ACTION ModeENLimk:
//屏蔽链接
Mach_Control.DT_b.FirstEmpFold:=par.iModeEN.FirstEmpFoldEN;				//首层空叠隔膜屏蔽
Mach_Control.DT_b.DP_Mode:=NOT par.iModeEN.DP_ModeEN;				//尾层空叠隔膜屏蔽
Mach_Control.DT_b.RectifydevModel:=par.iModeEN.RectifydevModelEN;			//隔膜纠偏屏蔽
Mach_Control.U.EmptyRunMode:=par.iModeEN.EmptyRunModeEN;				//空叠隔膜屏蔽
Mach_Control.U.CCD_ChosesHMI:=par.iModeEN.CCD_ChosesHMIEN;			//CCD屏蔽
Mach_Control.DT_b.DT_CCD_TwoModel:=NOT par.iModeEN.DT_CCD_TwoModelEN;		//CCD复检屏蔽
Mach_Control.DT_b.DT_Overhang:=par.iModeEN.DT_OverhangEN;				//对齐度屏蔽
Mach_Control.DT_b.DT_CellNG_TF:=NOT par.iModeEN.DT_CellNG_TFEN;				//对齐度踢废屏蔽 
Mach_Control.DT_b.DT_OHclosure:= par.iModeEN.DT_OHclosureEN;				//对齐度闭环屏蔽		ON是屏蔽
Mach_Control.DT_b.GMAngleALMsel:= par.iModeEN.GMAngleALMsel; //隔膜卷径报警屏蔽		ON是屏蔽
END_ACTION

ACTION MotionCoe_Write:

//nSlaveAddr :ARRAY[1..6] OF INT :=[1003,1008,1018,1019,1020,1021] ;     //EtherCAT支路驱动器ID

//'192.168.10.10.4.1'	EtherCat支路ID
(*
//隔膜平移地址
P2M1_Par.stDT_date.EtherCatAddr[1]:=1172;
P2M2_Par.stDT_date.EtherCatAddr[1]:=1123;
P2M3_Par.stDT_date.EtherCatAddr[1]:=1077;

//隔膜缓存地址
P2M1_Par.stDT_date.EtherCatAddr[2]:=1173;
P2M2_Par.stDT_date.EtherCatAddr[2]:=1124;
P2M3_Par.stDT_date.EtherCatAddr[2]:=1078;

//正极送片搬运平移地址
P2M1_Par.stDT_date.EtherCatAddr[3]:=1170;
P2M2_Par.stDT_date.EtherCatAddr[3]:=1121;
P2M3_Par.stDT_date.EtherCatAddr[3]:=1075;

//正极叠片搬运平移地址
P2M1_Par.stDT_date.EtherCatAddr[4]:=1171;
P2M2_Par.stDT_date.EtherCatAddr[4]:=1122;
P2M3_Par.stDT_date.EtherCatAddr[4]:=1076;

//负极送片搬运平移地址
P2M1_Par.stDT_date.EtherCatAddr[5]:=1188;
P2M2_Par.stDT_date.EtherCatAddr[5]:=1139;
P2M3_Par.stDT_date.EtherCatAddr[5]:=1093;

//负极叠片搬运平移地址
P2M1_Par.stDT_date.EtherCatAddr[6]:=1172;
P2M2_Par.stDT_date.EtherCatAddr[6]:=1140;
P2M3_Par.stDT_date.EtherCatAddr[6]:=1094;

//////////////////////////////////////////////////////////////////////一号叠台隔膜平移
FB_EcCoESdoWrite_SEPTATLine[1](
	sNetId:= '192.168.10.10.4.1', 
	nSlaveAddr:=Par.stDT_date.EtherCatAddr[1] ,   //隔膜平移
	nSubIndex:=0 , 
	nIndex:=16#2108 ,   //  平滑时间
	pSrcBuf:=ADR(Par.stDT_date.SEPTATLine_fSmoothValue[1]),       //写入参数值 
	cbBufLen:=SIZEOF(Par.stDT_date.SEPTATLine_fSmoothValue[1]),    
	bExecute:= Par.stDT_date.SEPTATLine_bWriteCoeValue[1],    
	tTimeout:= T#3S, 
	bBusy=> , 
	bError=> , 
	nErrId=> );
	
FB_EcCoESdoWrite_SEPTATLine[2](
	sNetId:='192.168.10.10.4.1', 
	nSlaveAddr:=Par.stDT_date.EtherCatAddr[1] ,   //隔膜平移
	nSubIndex:=0 , 
	nIndex:=16#2109 ,   // 平滑方式
	pSrcBuf:=ADR(Par.stDT_date.SEPTATLine_fSmoothValue[2]),       //写入参数值 
	cbBufLen:=SIZEOF(Par.stDT_date.SEPTATLine_fSmoothValue[2]),    
	bExecute:= Par.stDT_date.SEPTATLine_bWriteCoeValue[2],    
	tTimeout:= T#3S, 
	bBusy=> , 
	bError=> , 
	nErrId=> );

//平滑时间参数保存	
FB_EcCoESdoWrite_SEPTATLine[3](
	sNetId:= '192.168.10.10.4.1', 
	nSlaveAddr:=Par.stDT_date.EtherCatAddr[1] ,   //隔膜平移
	nSubIndex:=0 , 
	nIndex:=16#2108 ,   // 平滑时间
	pSrcBuf:=ADR(Par.stDT_date.wSaveCoeCode),      
	cbBufLen:=SIZEOF(Par.stDT_date.wSaveCoeCode),    
	bExecute:= Par.stDT_date.SEPTATLine_SavePara[1],    
	tTimeout:= T#3S, 
	bBusy=> , 
	bError=> , 
	nErrId=> );	
	
//平滑方式参数保存	
FB_EcCoESdoWrite_SEPTATLine[4](
	sNetId:= '192.168.10.10.4.1', 
	nSlaveAddr:=Par.stDT_date.EtherCatAddr[1] ,   //隔膜平移
	nSubIndex:=0 , 
	nIndex:=16#2109 ,   // 平滑方式
	pSrcBuf:=ADR(Par.stDT_date.wSaveCoeCode),      
	cbBufLen:=SIZEOF(Par.stDT_date.wSaveCoeCode),    
	bExecute:= Par.stDT_date.SEPTATLine_SavePara[2],    
	tTimeout:= T#3S, 
	bBusy=> , 
	bError=> , 
	nErrId=> );	

	
//////////////////////////////////////////////////////////////////////一号叠台隔膜缓存
FB_EcCoESdoWrite_SEPTATCache[1](
	sNetId:='192.168.10.10.4.1', 
	nSlaveAddr:=Par.stDT_date.EtherCatAddr[2] ,   //隔膜缓存
	nSubIndex:=0 , 
	nIndex:=16#2108 ,   //  平滑时间
	pSrcBuf:=ADR(Par.stDT_date.SEPTATCache_fSmoothValue[1]),       //写入参数值 
	cbBufLen:=SIZEOF(Par.stDT_date.SEPTATCache_fSmoothValue[1]),    
	bExecute:= Par.stDT_date.SEPTATCache_bWriteCoeValue[1],    
	tTimeout:= T#3S, 
	bBusy=> , 
	bError=> , 
	nErrId=> );
	
FB_EcCoESdoWrite_SEPTATCache[2](
	sNetId:='192.168.10.10.4.1', 
	nSlaveAddr:=Par.stDT_date.EtherCatAddr[2] ,   //隔膜缓存
	nSubIndex:=0 , 
	nIndex:=16#2109 ,   // 平滑方式
	pSrcBuf:=ADR(Par.stDT_date.SEPTATCache_fSmoothValue[2]),       //写入参数值 
	cbBufLen:=SIZEOF(Par.stDT_date.SEPTATCache_fSmoothValue[2]),    
	bExecute:= Par.stDT_date.SEPTATCache_bWriteCoeValue[2],    
	tTimeout:= T#3S, 
	bBusy=> , 
	bError=> , 
	nErrId=> );

//平滑时间参数保存	
FB_EcCoESdoWrite_SEPTATCache[3](
	sNetId:= '192.168.10.10.4.1', 
	nSlaveAddr:=Par.stDT_date.EtherCatAddr[2] ,   //隔膜缓存
	nSubIndex:=0 , 
	nIndex:=16#2108 ,   // 平滑时间
	pSrcBuf:=ADR(Par.stDT_date.wSaveCoeCode),      
	cbBufLen:=SIZEOF(Par.stDT_date.wSaveCoeCode),    
	bExecute:= Par.stDT_date.SEPTATCache_SavePara[1],    
	tTimeout:= T#3S, 
	bBusy=> , 
	bError=> , 
	nErrId=> );	
	
//平滑方式参数保存	
FB_EcCoESdoWrite_SEPTATCache[4](
	sNetId:= '192.168.10.10.4.1', 
	nSlaveAddr:=Par.stDT_date.EtherCatAddr[2] ,   //隔膜缓存
	nSubIndex:=0 , 
	nIndex:=16#2109 ,   // 平滑方式
	pSrcBuf:=ADR(Par.stDT_date.wSaveCoeCode),      
	cbBufLen:=SIZEOF(Par.stDT_date.wSaveCoeCode),    
	bExecute:= Par.stDT_date.SEPTATCache_SavePara[2],    
	tTimeout:= T#3S, 
	bBusy=> , 
	bError=> , 
	nErrId=> );	
	
	
//////////////////////////////////////////////////////////////////////正极送片搬运平移
FB_EcCoESdoWrite_AnCarryingLine[1](
	sNetId:= '192.168.10.10.4.1', 
	nSlaveAddr:=Par.stDT_date.EtherCatAddr[3] ,   //正极送片搬运平移
	nSubIndex:=0 , 
	nIndex:=16#2108 ,   //  平滑时间
	pSrcBuf:=ADR(Par.stDT_date.AnCarryingLine_fSmoothValue[1]),       //写入参数值 
	cbBufLen:=SIZEOF(Par.stDT_date.AnCarryingLine_fSmoothValue[1]),    
	bExecute:= Par.stDT_date.AnCarryingLine_bWriteCoeValue[1],    
	tTimeout:= T#3S, 
	bBusy=> , 
	bError=> , 
	nErrId=> );
	
FB_EcCoESdoWrite_AnCarryingLine[2](
	sNetId:= '192.168.10.10.4.1', 
	nSlaveAddr:=Par.stDT_date.EtherCatAddr[3]  ,   //正极送片搬运平移
	nSubIndex:=0 , 
	nIndex:=16#2109 ,   // 平滑方式
	pSrcBuf:=ADR(Par.stDT_date.AnCarryingLine_fSmoothValue[2]),       //写入参数值 
	cbBufLen:=SIZEOF(Par.stDT_date.AnCarryingLine_fSmoothValue[2]),    
	bExecute:= Par.stDT_date.AnCarryingLine_bWriteCoeValue[2],    
	tTimeout:= T#3S, 
	bBusy=> , 
	bError=> , 
	nErrId=> );

//平滑时间参数保存	
FB_EcCoESdoWrite_AnCarryingLine[3](
	sNetId:= '192.168.10.10.4.1', 
	nSlaveAddr:=Par.stDT_date.EtherCatAddr[3]  ,   //正极送片搬运平移
	nSubIndex:=0 , 
	nIndex:=16#2108 ,   // 平滑时间
	pSrcBuf:=ADR(Par.stDT_date.wSaveCoeCode),      
	cbBufLen:=SIZEOF(Par.stDT_date.wSaveCoeCode),    
	bExecute:= Par.stDT_date.AnCarryingLine_SavePara[1],    
	tTimeout:= T#3S, 
	bBusy=> , 
	bError=> , 
	nErrId=> );	
	
//平滑方式参数保存	
FB_EcCoESdoWrite_AnCarryingLine[4](
	sNetId:= '192.168.10.10.4.1', 
	nSlaveAddr:=Par.stDT_date.EtherCatAddr[3]  ,   //正极送片搬运平移
	nSubIndex:=0 , 
	nIndex:=16#2109 ,   // 平滑方式
	pSrcBuf:=ADR(Par.stDT_date.wSaveCoeCode),      
	cbBufLen:=SIZEOF(Par.stDT_date.wSaveCoeCode),    
	bExecute:= Par.stDT_date.AnCarryingLine_SavePara[2],    
	tTimeout:= T#3S, 
	bBusy=> , 
	bError=> , 
	nErrId=> );		
	
//////////////////////////////////////////////////////////////////////正极叠片搬运平移
FB_EcCoESdoWrite_AnDTCarryingLine[1](
	sNetId:='192.168.10.10.4.1', 
	nSlaveAddr:=Par.stDT_date.EtherCatAddr[4]  ,   //正极叠片搬运平移
	nSubIndex:=0 , 
	nIndex:=16#2108 ,   //  平滑时间
	pSrcBuf:=ADR(Par.stDT_date.AnDTCarryingLine_fSmoothValue[1]),       //写入参数值 
	cbBufLen:=SIZEOF(Par.stDT_date.AnDTCarryingLine_fSmoothValue[1]),    
	bExecute:= Par.stDT_date.AnDTCarryingLine_bWriteCoeValue[1],    
	tTimeout:= T#3S, 
	bBusy=> , 
	bError=> , 
	nErrId=> );
	
FB_EcCoESdoWrite_AnDTCarryingLine[2](
	sNetId:= '192.168.10.10.4.1', 
	nSlaveAddr:=Par.stDT_date.EtherCatAddr[4]  ,   //正极叠片搬运平移
	nSubIndex:=0 , 
	nIndex:=16#2109 ,   // 平滑方式
	pSrcBuf:=ADR(Par.stDT_date.AnDTCarryingLine_fSmoothValue[2]),       //写入参数值 
	cbBufLen:=SIZEOF(Par.stDT_date.AnDTCarryingLine_fSmoothValue[2]),    
	bExecute:= Par.stDT_date.AnDTCarryingLine_bWriteCoeValue[2],    
	tTimeout:= T#3S, 
	bBusy=> , 
	bError=> , 
	nErrId=> );

//平滑时间参数保存	
FB_EcCoESdoWrite_AnDTCarryingLine[3](
	sNetId:= '192.168.10.10.4.1', 
	nSlaveAddr:=Par.stDT_date.EtherCatAddr[4]  ,   //正极叠片搬运平移
	nSubIndex:=0 , 
	nIndex:=16#2108 ,   // 平滑时间
	pSrcBuf:=ADR(Par.stDT_date.wSaveCoeCode),      
	cbBufLen:=SIZEOF(Par.stDT_date.wSaveCoeCode),    
	bExecute:= Par.stDT_date.AnDTCarryingLine_SavePara[1],    
	tTimeout:= T#3S, 
	bBusy=> , 
	bError=> , 
	nErrId=> );	
	
//平滑方式参数保存	
FB_EcCoESdoWrite_AnDTCarryingLine[4](
	sNetId:= '192.168.10.10.4.1', 
	nSlaveAddr:=Par.stDT_date.EtherCatAddr[4]  ,   //正极叠片搬运平移
	nSubIndex:=0 , 
	nIndex:=16#2109 ,   // 平滑方式
	pSrcBuf:=ADR(Par.stDT_date.wSaveCoeCode),      
	cbBufLen:=SIZEOF(Par.stDT_date.wSaveCoeCode),    
	bExecute:= Par.stDT_date.AnDTCarryingLine_SavePara[2],    
	tTimeout:= T#3S, 
	bBusy=> , 
	bError=> , 
	nErrId=> );			
	
//////////////////////////////////////////////////////////////////////负极送片搬运平移
FB_EcCoESdoWrite_CaCarryingLine2[1](
	sNetId:= '192.168.10.10.4.1', 
	nSlaveAddr:=Par.stDT_date.EtherCatAddr[5]  ,   //负极送片搬运平移
	nSubIndex:=0 , 
	nIndex:=16#2108 ,   //  平滑时间
	pSrcBuf:=ADR(Par.stDT_date.CaCarryingLine2_fSmoothValue[1]),       //写入参数值 
	cbBufLen:=SIZEOF(Par.stDT_date.CaCarryingLine2_fSmoothValue[1]),    
	bExecute:= Par.stDT_date.CaCarryingLine2_bWriteCoeValue[1],    
	tTimeout:= T#3S, 
	bBusy=> , 
	bError=> , 
	nErrId=> );
	
FB_EcCoESdoWrite_CaCarryingLine2[2](
	sNetId:= '192.168.10.10.4.1', 
	nSlaveAddr:=Par.stDT_date.EtherCatAddr[5] ,   //负极送片搬运平移
	nSubIndex:=0 , 
	nIndex:=16#2109 ,   // 平滑方式
	pSrcBuf:=ADR(Par.stDT_date.CaCarryingLine2_fSmoothValue[2]),       //写入参数值 
	cbBufLen:=SIZEOF(Par.stDT_date.CaCarryingLine2_fSmoothValue[2]),    
	bExecute:= Par.stDT_date.CaCarryingLine2_bWriteCoeValue[2],    
	tTimeout:= T#3S, 
	bBusy=> , 
	bError=> , 
	nErrId=> );

//平滑时间参数保存	
FB_EcCoESdoWrite_CaCarryingLine2[3](
	sNetId:= '192.168.10.10.4.1', 
	nSlaveAddr:=Par.stDT_date.EtherCatAddr[5] ,   //负极送片搬运平移
	nSubIndex:=0 , 
	nIndex:=16#2108 ,   // 平滑时间
	pSrcBuf:=ADR(Par.stDT_date.wSaveCoeCode),      
	cbBufLen:=SIZEOF(Par.stDT_date.wSaveCoeCode),    
	bExecute:= Par.stDT_date.CaCarryingLine2_SavePara[1],    
	tTimeout:= T#3S, 
	bBusy=> , 
	bError=> , 
	nErrId=> );	
	
//平滑方式参数保存	
FB_EcCoESdoWrite_CaCarryingLine2[4](
	sNetId:='192.168.10.10.4.1', 
	nSlaveAddr:=Par.stDT_date.EtherCatAddr[5] ,   //负极送片搬运平移
	nSubIndex:=0 , 
	nIndex:=16#2109 ,   // 平滑方式
	pSrcBuf:=ADR(Par.stDT_date.wSaveCoeCode),      
	cbBufLen:=SIZEOF(Par.stDT_date.wSaveCoeCode),    
	bExecute:= Par.stDT_date.CaCarryingLine2_SavePara[2],    
	tTimeout:= T#3S, 
	bBusy=> , 
	bError=> , 
	nErrId=> );				
	
//////////////////////////////////////////////////////////////////////负极叠片搬运平移
FB_EcCoESdoWrite_CaDTCarryingLine[1](
	sNetId:= '192.168.10.10.4.1', 
	nSlaveAddr:=Par.stDT_date.EtherCatAddr[6]  ,   //负极叠片搬运平移
	nSubIndex:=0 , 
	nIndex:=16#2108 ,   //  平滑时间
	pSrcBuf:=ADR(Par.stDT_date.CaDTCarryingLine_fSmoothValue[1]),       //写入参数值 
	cbBufLen:=SIZEOF(Par.stDT_date.CaDTCarryingLine_fSmoothValue[1]),    
	bExecute:= Par.stDT_date.CaDTCarryingLine_bWriteCoeValue[1],    
	tTimeout:= T#3S, 
	bBusy=> , 
	bError=> , 
	nErrId=> );
	
FB_EcCoESdoWrite_CaDTCarryingLine[2](
	sNetId:= '192.168.10.10.4.1', 
	nSlaveAddr:=Par.stDT_date.EtherCatAddr[6]  ,   //负极叠片搬运平移
	nSubIndex:=0 , 
	nIndex:=16#2109 ,   // 平滑方式
	pSrcBuf:=ADR(Par.stDT_date.CaDTCarryingLine_fSmoothValue[2]),       //写入参数值 
	cbBufLen:=SIZEOF(Par.stDT_date.CaDTCarryingLine_fSmoothValue[2]),    
	bExecute:= Par.stDT_date.CaDTCarryingLine_bWriteCoeValue[2],    
	tTimeout:= T#3S, 
	bBusy=> , 
	bError=> , 
	nErrId=> );

//平滑时间参数保存	
FB_EcCoESdoWrite_CaDTCarryingLine[3](
	sNetId:= '192.168.10.10.4.1', 
	nSlaveAddr:=Par.stDT_date.EtherCatAddr[6]  ,   //负极叠片搬运平移
	nSubIndex:=0 , 
	nIndex:=16#2108 ,   // 平滑时间
	pSrcBuf:=ADR(Par.stDT_date.wSaveCoeCode),      
	cbBufLen:=SIZEOF(Par.stDT_date.wSaveCoeCode),    
	bExecute:= Par.stDT_date.CaDTCarryingLine_SavePara[1],    
	tTimeout:= T#3S, 
	bBusy=> , 
	bError=> , 
	nErrId=> );	
	
//平滑方式参数保存	
FB_EcCoESdoWrite_CaDTCarryingLine[4](
	sNetId:='192.168.10.10.4.1', 
	nSlaveAddr:=Par.stDT_date.EtherCatAddr[6]  ,   //负极叠片搬运平移
	nSubIndex:=0 , 
	nIndex:=16#2109 ,   // 平滑方式
	pSrcBuf:=ADR(Par.stDT_date.wSaveCoeCode),      
	cbBufLen:=SIZEOF(Par.stDT_date.wSaveCoeCode),    
	bExecute:= Par.stDT_date.CaDTCarryingLine_SavePara[2],    
	tTimeout:= T#3S, 
	bBusy=> , 
	bError=> , 
	nErrId=> );				
	*)
END_ACTION

ACTION P2_Init:
//上电初始化
	CASE Mach_Control.U.Step[0] OF 
			0://等待上电初始化启动
				IF Mach_Control.U.P2Init AND NOT Mach_Control.U.P2InitDone THEN
					Mach_Control.U.Step[0] :=10;
				END_IF
			10://气缸类型初始化,气控阀类型初始化
					//气缸类型初始化
					arrCyCtrl[arrCyNo.CylinderName.	AnScrapbinCy		].Cmd.iType:=	1	;//	正极片NG收纳盒
					arrCyCtrl[arrCyNo.CylinderName.	CaScrapbinCy		].Cmd.iType:=	1	;//	负极片NG收纳盒
					arrCyCtrl[arrCyNo.CylinderName.CaScrapbinUDCy		].Cmd.iType:=	1	;//	负极片NG收纳盒升降
					arrCyCtrl[arrCyNo.CylinderName.	PoleInflationCy		].Cmd.iType:=	3	;//	隔膜放卷气胀轴
					arrCyCtrl[arrCyNo.CylinderName.	PoleTapeSplicerLCy		].Cmd.iType:=	1	;//	隔膜接带左压板气缸
					arrCyCtrl[arrCyNo.CylinderName.	PoleTapeSplicerRCy		].Cmd.iType:=	1	;//	隔膜接带右压板气缸
					arrCyCtrl[arrCyNo.CylinderName.PreDiaph		].Cmd.iType:=	1	;//	叠台压隔膜气缸
					arrCyCtrl[arrCyNo.CylinderName.	PoleTapeCy		].Cmd.iType:=	1	;//	隔膜夹紧气缸
					arrCyCtrl[arrCyNo.CylinderName.	PoleHotCutterCy		].Cmd.iType:=	1	;//	隔膜热切升降
					arrCyCtrl[arrCyNo.CylinderName.	PoleSplintCy_U		].Cmd.iType:=	1	;//	夹膜上夹板
					arrCyCtrl[arrCyNo.CylinderName.	PoleSplintCy_D		].Cmd.iType:=	1	;//	夹膜下夹板
					arrCyCtrl[arrCyNo.CylinderName.	TailCurlSplintCy		].Cmd.iType:=	1	;//	尾卷夹爪开合
					arrCyCtrl[arrCyNo.CylinderName.	CurlingSplintCy_L		].Cmd.iType:=	3	;//	长卷针夹开合
					arrCyCtrl[arrCyNo.CylinderName.	CurlingSplintCy_S		].Cmd.iType:=	3	;//	短卷针夹开合
					//arrCyCtrl[arrCyNo.CylinderName.	CurlingSplintCy_S_1		].Cmd.iType:=	2	;//	短卷针夹开合_1
					arrCyCtrl[arrCyNo.CylinderName.	TailCurlLineCy		].Cmd.iType:=	1	;//	尾卷压辊平移缸
					arrCyCtrl[arrCyNo.CylinderName.	TailCurlUpdownCy		].Cmd.iType:=	1	;//	尾卷压辊升降缸
					arrCyCtrl[arrCyNo.CylinderName.	StandbyGlueCy		].Cmd.iType:=	2	;//	备胶气缸
					arrCyCtrl[arrCyNo.CylinderName.	CodeStandbyGlueCy		].Cmd.iType:=	2	;//	备二维码胶气缸
					arrCyCtrl[arrCyNo.CylinderName.	GlueClampsCy		].Cmd.iType:=	1	;//	贴胶夹爪气缸
					arrCyCtrl[arrCyNo.CylinderName.	GluePressCy		].Cmd.iType:=	1	;//	压胶气缸
					arrCyCtrl[arrCyNo.CylinderName.	CodeGluePressCy		].Cmd.iType:=	1	;//	压二维码胶气缸
					arrCyCtrl[arrCyNo.CylinderName.	GlueCutCy		].Cmd.iType:=	1	;//	切胶气缸
					arrCyCtrl[arrCyNo.CylinderName.	codeGlueCutCy		].Cmd.iType:=	1	;//	切二维码胶气缸
					arrCyCtrl[arrCyNo.CylinderName.	PullGluePoleCy		].Cmd.iType:=	4	;//	拉胶杆抱紧
					arrCyCtrl[arrCyNo.CylinderName.	PullGlueCy		].Cmd.iType:=	1	;//	拉胶气缸
					arrCyCtrl[arrCyNo.CylinderName.	GlueNGCy		].Cmd.iType:=	1	;//	踢废胶气缸
					arrCyCtrl[arrCyNo.CylinderName.	PullGlueModelCy		].Cmd.iType:=	1	;//	贴胶治具气缸
					//气控阀类型初始化				
					arrCyCtrl[arrCyNo.ElectValveName.	AnBeltVacuum		].Cmd.iType:=	4	;//	正极模切送料分段皮带1取料处真空
					arrCyCtrl[arrCyNo.ElectValveName.	AnBeltVacuumBark		].Cmd.iType:=	4	;//	正极模切送料分段皮带1取料处破真空
					arrCyCtrl[arrCyNo.ElectValveName.	CaMQBeltVacuum		].Cmd.iType:=	4	;//	负极模切送料分段皮带1取料处真空
					arrCyCtrl[arrCyNo.ElectValveName.	CaMQBeltVacuumBark		].Cmd.iType:=	4	;//	负极模切送料分段皮带1取料处破真空
					arrCyCtrl[arrCyNo.ElectValveName.	AnCarryingVacuum		].Cmd.iType:=	4	;//	正极送片搬运升降真空
					arrCyCtrl[arrCyNo.ElectValveName.	AnCarryingVacuumBark		].Cmd.iType:=	4	;//	正极送片搬运升降破真空
					arrCyCtrl[arrCyNo.ElectValveName.	AndeviationVacuum		].Cmd.iType:=	4	;//	正极纠偏平台真空
					arrCyCtrl[arrCyNo.ElectValveName.	AndeviationIonizedWind		].Cmd.iType:=	4	;//	正极纠偏平台除尘风刀
					arrCyCtrl[arrCyNo.ElectValveName.	AndeviationVacuumBark		].Cmd.iType:=	4	;//	正极纠偏平台破真空
					arrCyCtrl[arrCyNo.ElectValveName.	AnDTCarryingVacuum		].Cmd.iType:=	4	;//	正极叠片搬运升降真空
					//arrCyCtrl[arrCyNo.ElectValveName.	AnDTCarryingJRVacuum		].Cmd.iType:=	4	;//	正极叠台搬运升降极耳真空
					arrCyCtrl[arrCyNo.ElectValveName.	AnDTCarryingVacuumBark		].Cmd.iType:=	4	;//	正极叠片搬运升降破真空
					arrCyCtrl[arrCyNo.ElectValveName.	CaCarryingVacuum1		].Cmd.iType:=	4	;//	负极送片搬运升降1真空
					arrCyCtrl[arrCyNo.ElectValveName.	CaCarryingVacuumBark1		].Cmd.iType:=	4	;//	负极送片搬运升降1破真空
					arrCyCtrl[arrCyNo.ElectValveName.	CaLoadUpBeltVacuum		].Cmd.iType:=	4	;//	负极送片皮带末端真空
					arrCyCtrl[arrCyNo.ElectValveName.	CaLoadUpBeltVacuumBark		].Cmd.iType:=	4	;//	负极送片皮带末端破真空
					arrCyCtrl[arrCyNo.ElectValveName.	CaCarryingVacuum2		].Cmd.iType:=	4	;//	负极送片搬运升降2真空
					arrCyCtrl[arrCyNo.ElectValveName.	CaCarryingVacuumBark2		].Cmd.iType:=	4	;//	负极送片搬运升降2破真空
					arrCyCtrl[arrCyNo.ElectValveName.	CadeviationVacuum		].Cmd.iType:=	4	;//	负极纠偏平台真空
					arrCyCtrl[arrCyNo.ElectValveName.	CadeviationVacuumBark		].Cmd.iType:=	4	;//	负极纠偏平台破真空
					arrCyCtrl[arrCyNo.ElectValveName.	CadeviationIonizedWind		].Cmd.iType:=	4	;//	负极纠偏平台除尘风刀
					arrCyCtrl[arrCyNo.ElectValveName.	CaDTCarryingVacuum		].Cmd.iType:=	4	;//	负极叠片搬运升降真空
					//arrCyCtrl[arrCyNo.ElectValveName.	CaDTCarryingJRVacuum		].Cmd.iType:=	4	;//	负极叠片搬运升降极耳真空
					arrCyCtrl[arrCyNo.ElectValveName.	CaDTCarryingVacuumBark		].Cmd.iType:=	4	;//	负极叠片搬运升降破真空
					arrCyCtrl[arrCyNo.ElectValveName.	PoleTapeDustRemoval		].Cmd.iType:=	4	;//	隔膜接带平台除尘
					arrCyCtrl[arrCyNo.ElectValveName.	PoleTapeVacuum		].Cmd.iType:=	4	;//	隔膜接带平台真空
					arrCyCtrl[arrCyNo.ElectValveName.	BlueGlueVacuum1		].Cmd.iType:=	4	;//	备胶组件蓝胶真空1
					arrCyCtrl[arrCyNo.ElectValveName.	BlueGlueVacuum2		].Cmd.iType:=	4	;//	备胶组件蓝胶真空2
					arrCyCtrl[arrCyNo.ElectValveName.	codeGlueVacuum1		].Cmd.iType:=	4	;//	备胶组件二维码胶真空1
					arrCyCtrl[arrCyNo.ElectValveName.	codeGlueVacuum2		].Cmd.iType:=	4	;//	备胶组件二维码胶真空2
					arrCyCtrl[arrCyNo.ElectValveName.	PastesGlueVacuum		].Cmd.iType:=	4	;//	备胶组件贴胶头真空
					arrCyCtrl[arrCyNo.ElectValveName.	DTVacuum		].Cmd.iType:=	4	;//	叠片台真空
					arrCyCtrl[arrCyNo.ElectValveName.	PoleSplintVacuum_D		].Cmd.iType:=	4	;//	夹膜下夹板真空
					arrCyCtrl[arrCyNo.ElectValveName.WJ_blow		].Cmd.iType:=	4	;//	夹电芯吹气
					arrCyCtrl[arrCyNo.ElectValveName.WJShortvacuum		].Cmd.iType:=	4	;//短卷针张开真空
					//屏蔽初赋值					
					Mach_Control.U.Step[0] :=20;
					
			20://计算从左到右、从右到左移动时隔膜变化量
					CaCrectCamStep0:=10;//负极取片凸轮创建
					AnCrectCamStep0:=10;//正极取片凸轮创建
					YDCrectCamStep0:=10;//叠台压刀凸轮创建
					GMCreatCamStep0:=10;//叠台缓存凸轮创建
					WZCreatCamStep0:=10;//尾卷凸轮创建
					Mach_Control.U.Step[0] :=30;
			30://判断隔膜变数据是否完成
					IF CaCrectCamStep0=6666 AND AnCrectCamStep0=6666 AND YDCrectCamStep0=6666 AND  GMCreatCamStep0=6666 AND WZCreatCamStep0=6666 THEN
						Mach_Control.U.Step[0] :=40;
					END_IF;
			40:
				arrCyCtrl[arrCyNo.CylinderName.PoleInflationCy].Cmd.bON:=TRUE;
				Mach_Control.U.P2Init :=FALSE;//复位上电初始化完成
				Mach_Control.U.P2InitDone:=TRUE;//置位上电初始化完成
				Mach_Control.U.Step[0] :=0;
	END_CASE

	arrCyCtrl[arrCyNo.ElectValveName.	CaCarryingVacuumBark2		].Cmd.bON;
END_ACTION

ACTION Stick_Condition:
//贴胶平移，贴胶旋转轴移动允许  AND  arrAxisCtrl[AxiseNo.AxisName.TailCurlLine].Status.fSetPos>=arrAxisPar[AxiseNo.AxisName.TailCurlLine].arrTargetPoint[1]+0.2 AND arrAxisPar[AxiseNo.AxisName.TailCurlWhirling].arrTargetPoint[1] 
IF arrAxisCtrl[AxiseNo.AxisName.GluingRetracting].Status.Homed 
AND arrAxisCtrl[AxiseNo.AxisName.GluingRetracting].Status.NoMoving 
AND arrAxisCtrl[AxiseNo.AxisName.GluingRetracting].Cmd.arrbRealPoint[1] 
AND  ((arrAxisCtrl[AxiseNo.AxisName.TailCurlLine].Status.fSetPos>=arrAxisPar[AxiseNo.AxisName.TailCurlLine].arrTargetPoint[1]-1 AND  arrAxisCtrl[AxiseNo.AxisName.TailCurlRetracting].Status.fSetPos<=arrAxisPar[AxiseNo.AxisName.TailCurlRetracting].arrTargetPoint[1]+1) OR
		 arrAxisCtrl[AxiseNo.AxisName.TailCurlWhirling].Cmd.arrbRealPoint[1]  )
AND  ((DTselect=1 AND (arrAxisCtrl[P3AxisNo.P3M1_ColdpreLine].Status.fActPos <=  arrAxisPar[P3AxisNo.P3M1_ColdpreLine].arrTargetPoint[2]-300 OR 
            arrAxisCtrl[P3AxisNo.P3M1_ColdpreLine].Status.fActPos >=  arrAxisPar[P3AxisNo.P3M1_ColdpreLine].arrTargetPoint[2]+300)) OR    
         (DTselect=2 AND (arrAxisCtrl[P3AxisNo.P3M1_ColdpreLine].Status.fActPos <=  arrAxisPar[P3AxisNo.P3M1_ColdpreLine].arrTargetPoint[3]-300 OR 
			 arrAxisCtrl[P3AxisNo.P3M1_ColdpreLine].Status.fActPos >=  arrAxisPar[P3AxisNo.P3M1_ColdpreLine].arrTargetPoint[3]+300)) OR
		 (DTselect=3 AND (arrAxisCtrl[P3AxisNo.P3M1_ColdpreLine].Status.fActPos <=  arrAxisPar[P3AxisNo.P3M1_ColdpreLine].arrTargetPoint[4]-300 OR 
			 arrAxisCtrl[P3AxisNo.P3M1_ColdpreLine].Status.fActPos >=  arrAxisPar[P3AxisNo.P3M1_ColdpreLine].arrTargetPoint[4]+300))  OR 
		( arrAxisCtrl[P3AxisNo.P3M1_ColdpreWhirling].Cmd.arrbRealPoint[1] OR arrAxisCtrl[P3AxisNo.P3M1_ColdpreWhirling].Cmd.arrbRealPoint[5] OR arrAxisCtrl[P3AxisNo.P3M1_ColdpreWhirling].Cmd.arrbRealPoint[6]) )
(*AND arrAxisCtrl[AxiseNo.AxisName.TailCurlLine].Status.Homed 
AND  arrAxisCtrl[AxiseNo.AxisName.TailCurlRetracting].Cmd.arrbRealPoint[1] 
AND arrAxisCtrl[AxiseNo.AxisName.TailCurlRetracting].Status.Homed 
AND(((arrAxisCtrl[AxiseNo.AxisName.TailCurlLine].Status.fSetPos>= (arrAxisPar[AxiseNo.AxisName.TailCurlLine].arrTargetPoint[1]-1) 
AND (arrAxisCtrl[AxiseNo.AxisName.TailCurlWhirling].Cmd.arrbRealPoint[1] 
OR arrAxisCtrl[AxiseNo.AxisName.TailCurlWhirling].Cmd.arrbRealPoint[3] 
OR  arrAxisCtrl[AxiseNo.AxisName.TailCurlWhirling].Cmd.arrbRealPoint[4])) 
OR((arrAxisCtrl[AxiseNo.AxisName.TailCurlLine].Status.fSetPos>= (arrAxisPar[AxiseNo.AxisName.TailCurlLine].arrTargetPoint[5]-1)) 
AND arrAxisCtrl[AxiseNo.AxisName.TailCurlWhirling].Cmd.arrbRealPoint[2])))*)    THEN
	arrAxisCtrl[AxiseNo.AxisName.GluingLine].Cmd.GoPoint_Condition[0]:=TRUE;
	GluingLineagree:=TRUE;//侧贴胶平移轴、侧贴胶旋转轴动作允许
ELSE
	GluingLineagree:=FALSE;
	arrAxisCtrl[AxiseNo.AxisName.GluingLine].Cmd.GoPoint_Condition[0]:=FALSE;
END_IF


//贴胶旋转轴移动允许
IF GluingLineagree THEN
	GluingWhirlingagree:=TRUE;//侧贴胶平移轴、侧贴胶旋转轴动作允许
ELSE
	GluingWhirlingagree:=FALSE;
END_IF


Mach_Control.TJ_b.WhirlingSafe:=(*arrAxisCtrl[AxiseNo.AxisName.GluingWhirling].Status.Homed AND arrAxisCtrl[AxiseNo.AxisName.GluingWhirling].Status.NoMoving
                        AND*) arrAxisCtrl[AxiseNo.AxisName.GluingRetracting].Status.Homed AND arrAxisCtrl[AxiseNo.AxisName.GluingRetracting].Cmd.arrbRealPoint[1]
						AND (arrAxisCtrl[AxiseNo.AxisName.GluingLine].Status.fActPos <= (arrAxisPar[AxiseNo.AxisName.GluingLine].arrTargetPoint[10]+1)) AND
                         ((DTselect=1 AND (arrAxisCtrl[P3AxisNo.P3M1_ColdpreLine].Status.fActPos <=  arrAxisPar[P3AxisNo.P3M1_ColdpreLine].arrTargetPoint[2]-300 OR 
                              arrAxisCtrl[P3AxisNo.P3M1_ColdpreLine].Status.fActPos >=  arrAxisPar[P3AxisNo.P3M1_ColdpreLine].arrTargetPoint[2]+300)) OR
						(DTselect=2 AND (arrAxisCtrl[P3AxisNo.P3M1_ColdpreLine].Status.fActPos <=  arrAxisPar[P3AxisNo.P3M1_ColdpreLine].arrTargetPoint[3]-300 OR 
													  arrAxisCtrl[P3AxisNo.P3M1_ColdpreLine].Status.fActPos >=  arrAxisPar[P3AxisNo.P3M1_ColdpreLine].arrTargetPoint[3]+300)) OR
						(DTselect=3 AND (arrAxisCtrl[P3AxisNo.P3M1_ColdpreLine].Status.fActPos <=  arrAxisPar[P3AxisNo.P3M1_ColdpreLine].arrTargetPoint[4]-300 OR 
													  arrAxisCtrl[P3AxisNo.P3M1_ColdpreLine].Status.fActPos >=  arrAxisPar[P3AxisNo.P3M1_ColdpreLine].arrTargetPoint[4]+300))  OR 
						 ( arrAxisCtrl[P3AxisNo.P3M1_ColdpreWhirling].Cmd.arrbRealPoint[1] OR arrAxisCtrl[P3AxisNo.P3M1_ColdpreWhirling].Cmd.arrbRealPoint[5] OR arrAxisCtrl[P3AxisNo.P3M1_ColdpreWhirling].Cmd.arrbRealPoint[6]) );

					//AND (arrAxisCtrl[AxiseNo.AxisName.GluingLine].Status.fSetPos >= (arrAxisPar[AxiseNo.AxisName.GluingLine].arrTargetPoint[10]-1));

//侧贴胶平移运动允许
arrAxisCtrl[AxiseNo.AxisName.GluingLine].Cmd.GoPoint_Condition[0]:=GluingLineagree OR Mach_Control.TJ_b.AxisConditionEN ;
arrAxisCtrl[AxiseNo.AxisName.GluingLine].Cmd.GoPoint_Condition[1]:=GluingLineagree OR Mach_Control.TJ_b.AxisConditionEN ;
//侧贴胶旋转运动允许
arrAxisCtrl[AxiseNo.AxisName.GluingWhirling].Cmd.GoPoint_Condition[0]:=GluingLineagree OR Mach_Control.TJ_b.AxisConditionEN ;
arrAxisCtrl[AxiseNo.AxisName.GluingWhirling].Cmd.GoPoint_Condition[1]:=GluingLineagree OR Mach_Control.TJ_b.AxisConditionEN ;


//侧贴胶平移、旋转在下料位，侧贴胶夹爪气缸张开，允许尾卷下电芯
IF arrAxisCtrl[AxiseNo.AxisName.GluingLine].Status.Homed AND arrAxisCtrl[AxiseNo.AxisName.GluingLine].Status.NoMoving AND arrAxisCtrl[AxiseNo.AxisName.GluingLine].Cmd.arrbRealPoint[1] AND 
	 arrAxisCtrl[AxiseNo.AxisName.GluingWhirling].Status.Homed AND arrAxisCtrl[AxiseNo.AxisName.GluingWhirling].Status.NoMoving AND arrAxisCtrl[AxiseNo.AxisName.GluingWhirling].Cmd.arrbRealPoint[1] AND
	arrCyCtrl[arrCyNo.CylinderName.GlueClampsCy].Io.DIOnSwitch THEN
	Mach_Control.TJ_b.Stickerragree:=TRUE;	
ELSE
	Mach_Control.TJ_b.Stickerragree:=FALSE;		
END_IF
//贴胶完成，允许冷压取电芯
IF Mach_Control.TJ_b.StickerDone AND Mach_Control.TJ_b.StickerFlag AND arrAxisCtrl[AxiseNo.AxisName.GluingLine].Cmd.arrbRealPoint[2] AND arrAxisCtrl[AxiseNo.AxisName.GluingWhirling].Cmd.arrbRealPoint[2]  THEN
	Mach_Control.TJ_b.StickerOffloading:=TRUE;
ELSE
	Mach_Control.TJ_b.StickerOffloading:=FALSE; 	
END_IF
//拉胶在安全位，允许贴胶头前进、后退
IF arrAxisCtrl[AxiseNo.AxisName.GluingUpDown].Status.Homed AND arrAxisCtrl[AxiseNo.AxisName.GluingUpDown].Status.NoMoving AND 
	(arrAxisCtrl[AxiseNo.AxisName.GluingUpDown].Status.fActPos<= arrAxisPar[AxiseNo.AxisName.GluingUpDown].arrTargetPoint[4] OR
	arrAxisCtrl[AxiseNo.AxisName.GluingUpDown].Status.fActPos>= arrAxisPar[AxiseNo.AxisName.GluingUpDown].arrTargetPoint[2]) 
	AND arrCyCtrl[arrCyNo.CylinderName.GlueClampsCy].Status.OFFState THEN
	GluingRetractingagree:=TRUE;//贴胶头前进轴动作允许
ELSE
	GluingRetractingagree:=FALSE;
END_IF

arrAxisCtrl[AxiseNo.AxisName.GluingRetracting].Cmd.GoPoint_Condition[0]:=GluingRetractingagree OR Mach_Control.TJ_b.AxisConditionEN ;
arrAxisCtrl[AxiseNo.AxisName.GluingRetracting].Cmd.GoPoint_Condition[1]:=GluingRetractingagree OR Mach_Control.TJ_b.AxisConditionEN ;
arrAxisCtrl[AxiseNo.AxisName.GluingRetracting].Cmd.GoPoint_Condition[2]:=GluingRetractingagree OR Mach_Control.TJ_b.AxisConditionEN ;
arrAxisCtrl[AxiseNo.AxisName.GluingRetracting].Cmd.GoPoint_Condition[3]:=GluingRetractingagree OR Mach_Control.TJ_b.AxisConditionEN ;
arrAxisCtrl[AxiseNo.AxisName.GluingRetracting].Cmd.GoPoint_Condition[4]:=GluingRetractingagree OR Mach_Control.TJ_b.AxisConditionEN ;
arrAxisCtrl[AxiseNo.AxisName.GluingRetracting].Cmd.GoPoint_Condition[5]:=GluingRetractingagree OR Mach_Control.TJ_b.AxisConditionEN ;
//拉胶升降允许动作
IF arrAxisCtrl[AxiseNo.AxisName.GluingRetracting].Status.Homed AND 
	arrAxisCtrl[AxiseNo.AxisName.GluingRetracting].Status.fActPos<= arrAxisPar[AxiseNo.AxisName.GluingRetracting].arrTargetPoint[1]+0.2 AND 
	arrCyCtrl[arrCyNo.CylinderName.codeGlueCutCy].Status.ONState AND
	arrCyCtrl[arrCyNo.CylinderName.GlueCutCy].Status.ONState AND
	arrCyCtrl[arrCyNo.CylinderName.GlueNGCy].Status.OFFState AND 
	arrCyCtrl[arrCyNo.CylinderName.PullGlueCy].Status.ONState  THEN
	GluingUpDownagree:=TRUE; 
ELSE
	GluingUpDownagree:=false;	
END_IF
arrAxisCtrl[AxiseNo.AxisName.GluingUpDown].Cmd.GoPoint_Condition[1]:=GluingUpDownagree OR Mach_Control.TJ_b.AxisConditionEN ;	
arrAxisCtrl[AxiseNo.AxisName.GluingUpDown].Cmd.GoPoint_Condition[2]:=GluingUpDownagree OR Mach_Control.TJ_b.AxisConditionEN ;	
arrAxisCtrl[AxiseNo.AxisName.GluingUpDown].Cmd.GoPoint_Condition[3]:=GluingUpDownagree OR Mach_Control.TJ_b.AxisConditionEN ;	
arrAxisCtrl[AxiseNo.AxisName.GluingUpDown].Cmd.GoPoint_Condition[4]:=GluingUpDownagree OR Mach_Control.TJ_b.AxisConditionEN ;	
arrAxisCtrl[AxiseNo.AxisName.GluingUpDown].Cmd.GoPoint_Condition[5]:=GluingUpDownagree OR Mach_Control.TJ_b.AxisConditionEN ;	
arrAxisCtrl[AxiseNo.AxisName.GluingUpDown].Cmd.GoPoint_Condition[6]:=GluingUpDownagree OR Mach_Control.TJ_b.AxisConditionEN ;	
arrAxisCtrl[AxiseNo.AxisName.GluingUpDown].Cmd.GoPoint_Condition[7]:=GluingUpDownagree OR Mach_Control.TJ_b.AxisConditionEN ;	
arrAxisCtrl[AxiseNo.AxisName.GluingUpDown].Cmd.GoPoint_Condition[8]:=GluingUpDownagree OR Mach_Control.TJ_b.AxisConditionEN ;	


//气缸条件
IF arrCyCtrl[arrCyNo.CylinderName.GlueCutCy].Status.OFFState AND arrCyCtrl[arrCyNo.CylinderName.GlueCutCy].Status.OFFState  THEN
	arrCyCtrl[arrCyNo.CylinderName.GlueNGCy].Cmd.OnCondition:=TRUE;
ELSE
	arrCyCtrl[arrCyNo.CylinderName.GlueNGCy].Cmd.OnCondition:=FALSE;
END_IF

/////////////////////////////////////////////////////////////
/////////////////////////////////////////////////////////
////////////////////////////////////////////电机条件
//侧贴胶平移
IF  Mach_Control.U.WJ_iMode=3 
  AND GluingLineagree
 OR Mach_Control.TJ_b.AxisConditionEN THEN
	arrAxisCtrl[AxiseNo.AxisName.GluingLine].Cmd.Home_Condition:=TRUE;
ELSE
	arrAxisCtrl[AxiseNo.AxisName.GluingLine].Cmd.Home_Condition:=FALSE;	
END_IF

IF  Mach_Control.U.WJ_iMode=3 
AND arrAxisCtrl[AxiseNo.AxisName.GluingLine].Status.Homed 
AND GluingLineagree
 OR Mach_Control.TJ_b.AxisConditionEN THEN
	arrAxisCtrl[AxiseNo.AxisName.GluingLine].Cmd.GoPoint_Condition[1]:=TRUE;
ELSE
	arrAxisCtrl[AxiseNo.AxisName.GluingLine].Cmd.GoPoint_Condition[1]:=FALSE;	
END_IF

IF  Mach_Control.U.WJ_iMode=3 
AND arrAxisCtrl[AxiseNo.AxisName.GluingLine].Status.Homed 
AND GluingLineagree
 OR Mach_Control.TJ_b.AxisConditionEN THEN
	arrAxisCtrl[AxiseNo.AxisName.GluingLine].Cmd.GoPoint_Condition[2]:=TRUE;
ELSE
	arrAxisCtrl[AxiseNo.AxisName.GluingLine].Cmd.GoPoint_Condition[2]:=FALSE;	
END_IF

IF  Mach_Control.U.WJ_iMode=3 
AND arrAxisCtrl[AxiseNo.AxisName.GluingLine].Status.Homed 
AND GluingLineagree
 OR Mach_Control.TJ_b.AxisConditionEN THEN
	arrAxisCtrl[AxiseNo.AxisName.GluingLine].Cmd.GoPoint_Condition[3]:=TRUE;
ELSE
	arrAxisCtrl[AxiseNo.AxisName.GluingLine].Cmd.GoPoint_Condition[3]:=FALSE;	
END_IF

IF  Mach_Control.U.WJ_iMode=3 
AND arrAxisCtrl[AxiseNo.AxisName.GluingLine].Status.Homed 
AND GluingLineagree
 OR Mach_Control.TJ_b.AxisConditionEN THEN
	arrAxisCtrl[AxiseNo.AxisName.GluingLine].Cmd.GoPoint_Condition[4]:=TRUE;
ELSE
	arrAxisCtrl[AxiseNo.AxisName.GluingLine].Cmd.GoPoint_Condition[4]:=FALSE;	
END_IF

IF  Mach_Control.U.WJ_iMode=3 
AND arrAxisCtrl[AxiseNo.AxisName.GluingLine].Status.Homed  
AND GluingLineagree
 OR Mach_Control.TJ_b.AxisConditionEN THEN
	arrAxisCtrl[AxiseNo.AxisName.GluingLine].Cmd.GoPoint_Condition[5]:=TRUE;
ELSE
	arrAxisCtrl[AxiseNo.AxisName.GluingLine].Cmd.GoPoint_Condition[5]:=FALSE;	
END_IF

IF  Mach_Control.U.WJ_iMode=3 
AND arrAxisCtrl[AxiseNo.AxisName.GluingLine].Status.Homed  
AND GluingLineagree
 OR Mach_Control.TJ_b.AxisConditionEN THEN
	arrAxisCtrl[AxiseNo.AxisName.GluingLine].Cmd.GoPoint_Condition[6]:=TRUE;
ELSE
	arrAxisCtrl[AxiseNo.AxisName.GluingLine].Cmd.GoPoint_Condition[6]:=FALSE;	
END_IF

IF  Mach_Control.U.WJ_iMode=3 
AND arrAxisCtrl[AxiseNo.AxisName.GluingLine].Status.Homed 
AND GluingLineagree
OR Mach_Control.TJ_b.AxisConditionEN THEN
	arrAxisCtrl[AxiseNo.AxisName.GluingLine].Cmd.GoPoint_Condition[8]:=TRUE;
ELSE
	arrAxisCtrl[AxiseNo.AxisName.GluingLine].Cmd.GoPoint_Condition[8]:=FALSE;	
END_IF

IF  Mach_Control.U.WJ_iMode=3 
AND arrAxisCtrl[AxiseNo.AxisName.GluingLine].Status.Homed 
AND GluingLineagree
OR Mach_Control.TJ_b.AxisConditionEN  THEN
	arrAxisCtrl[AxiseNo.AxisName.GluingLine].Cmd.GoPoint_Condition[9]:=TRUE;
ELSE
	arrAxisCtrl[AxiseNo.AxisName.GluingLine].Cmd.GoPoint_Condition[9]:=FALSE;	
END_IF

IF  Mach_Control.U.WJ_iMode=3 
AND arrAxisCtrl[AxiseNo.AxisName.GluingLine].Status.Homed 
AND GluingLineagree
 OR Mach_Control.TJ_b.AxisConditionEN THEN
	arrAxisCtrl[AxiseNo.AxisName.GluingLine].Cmd.GoPoint_Condition[10]:=TRUE;
ELSE
	arrAxisCtrl[AxiseNo.AxisName.GluingLine].Cmd.GoPoint_Condition[10]:=FALSE;	
END_IF

//侧贴胶旋转//暂时屏蔽冷压
IF  Mach_Control.U.WJ_iMode=3 
//AND arrAxisCtrl[AxiseNo.AxisName.GluingWhirling].Status.Homed  
AND Mach_Control.TJ_b.WhirlingSafe
OR Mach_Control.TJ_b.AxisConditionEN THEN
	arrAxisCtrl[AxiseNo.AxisName.GluingWhirling].Cmd.Home_Condition:=TRUE;
ELSE
	arrAxisCtrl[AxiseNo.AxisName.GluingWhirling].Cmd.Home_Condition:=FALSE;	
END_IF

IF  Mach_Control.U.WJ_iMode=3 
AND arrAxisCtrl[AxiseNo.AxisName.GluingWhirling].Status.Homed  
AND arrAxisCtrl[AxiseNo.AxisName.GluingRetracting].Cmd.arrbRealPoint[1] 
AND ((arrAxisCtrl[AxiseNo.AxisName.TailCurlLine].Status.fSetPos>=arrAxisPar[AxiseNo.AxisName.TailCurlLine].arrTargetPoint[10]-1 
AND  arrAxisCtrl[AxiseNo.AxisName.TailCurlRetracting].Status.fSetPos<=arrAxisPar[AxiseNo.AxisName.TailCurlRetracting].arrTargetPoint[1]+1) OR arrAxisCtrl[AxiseNo.AxisName.TailCurlWhirling].Cmd.arrbRealPoint[1]) 
AND ((arrAxisCtrl[P3AxisNo.P3M1_ColdpreWhirling].Cmd.arrbRealPoint[1] 
OR arrAxisCtrl[P3AxisNo.P3M1_ColdpreWhirling].Cmd.arrbRealPoint[5]
OR arrAxisCtrl[P3AxisNo.P3M1_ColdpreWhirling].Cmd.arrbRealPoint[6] ) 
(*OR arrAxisCtrl[P3AxisNo.P3M1_ColdpreRetracting].Cmd.arrbRealPoint[1]*))
AND NOT arrAxisCtrl[AxiseNo.AxisName.GluingLine].Cmd.arrbRealPoint[8]
OR Mach_Control.TJ_b.AxisConditionEN THEN
	arrAxisCtrl[AxiseNo.AxisName.GluingWhirling].Cmd.GoPoint_Condition[1]:=TRUE;
	arrAxisCtrl[AxiseNo.AxisName.GluingWhirling].Cmd.GoPoint_Condition[2]:=TRUE;
	arrAxisCtrl[AxiseNo.AxisName.GluingWhirling].Cmd.GoPoint_Condition[3]:=TRUE;
	arrAxisCtrl[AxiseNo.AxisName.GluingWhirling].Cmd.GoPoint_Condition[4]:=TRUE;
	arrAxisCtrl[AxiseNo.AxisName.GluingWhirling].Cmd.GoPoint_Condition[5]:=TRUE;
	arrAxisCtrl[AxiseNo.AxisName.GluingWhirling].Cmd.GoPoint_Condition[6]:=TRUE;
ELSE
	arrAxisCtrl[AxiseNo.AxisName.GluingWhirling].Cmd.GoPoint_Condition[1]:=FALSE;
	arrAxisCtrl[AxiseNo.AxisName.GluingWhirling].Cmd.GoPoint_Condition[2]:=FALSE;
	arrAxisCtrl[AxiseNo.AxisName.GluingWhirling].Cmd.GoPoint_Condition[3]:=FALSE;
	arrAxisCtrl[AxiseNo.AxisName.GluingWhirling].Cmd.GoPoint_Condition[4]:=TRUE;
	arrAxisCtrl[AxiseNo.AxisName.GluingWhirling].Cmd.GoPoint_Condition[5]:=FALSE;
	arrAxisCtrl[AxiseNo.AxisName.GluingWhirling].Cmd.GoPoint_Condition[6]:=FALSE;	
END_IF
(*
IF  Mach_Control.U.WJ_iMode=3 AND arrAxisCtrl[AxiseNo.AxisName.GluingWhirling].Status.Homed  AND arrAxisCtrl[AxiseNo.AxisName.GluingRetracting].Cmd.arrbRealPoint[1] 
AND  ((arrAxisCtrl[AxiseNo.AxisName.TailCurlLine].Status.fSetPos>=arrAxisPar[AxiseNo.AxisName.TailCurlLine].arrTargetPoint[1]-1 AND  arrAxisCtrl[AxiseNo.AxisName.TailCurlRetracting].Status.fSetPos<=arrAxisPar[AxiseNo.AxisName.TailCurlRetracting].arrTargetPoint[1]+1) OR
    	  arrAxisCtrl[AxiseNo.AxisName.TailCurlWhirling].Cmd.arrbRealPoint[1]  ) 
 AND  ( (  arrAxisCtrl[P3AxisNo.P3M1_ColdpreWhirling].Cmd.arrbRealPoint[1] OR arrAxisCtrl[P3AxisNo.P3M1_ColdpreWhirling].Cmd.arrbRealPoint[5] OR arrAxisCtrl[P3AxisNo.P3M1_ColdpreWhirling].Cmd.arrbRealPoint[6] ) OR
                    arrAxisCtrl[P3AxisNo.P3M1_ColdpreRetracting].Cmd.arrbRealPoint[1] )
 OR Mach_Control.TJ_b.AxisConditionEN THEN
	arrAxisCtrl[AxiseNo.AxisName.GluingWhirling].Cmd.GoPoint_Condition[2]:=TRUE;
ELSE
	arrAxisCtrl[AxiseNo.AxisName.GluingWhirling].Cmd.GoPoint_Condition[2]:=FALSE;	
END_IF

IF  Mach_Control.U.WJ_iMode=3 AND arrAxisCtrl[AxiseNo.AxisName.GluingWhirling].Status.Homed  AND arrAxisCtrl[AxiseNo.AxisName.GluingRetracting].Cmd.arrbRealPoint[1] 
AND  ((arrAxisCtrl[AxiseNo.AxisName.TailCurlLine].Status.fSetPos>=arrAxisPar[AxiseNo.AxisName.TailCurlLine].arrTargetPoint[1]-1 AND  arrAxisCtrl[AxiseNo.AxisName.TailCurlRetracting].Status.fSetPos<=arrAxisPar[AxiseNo.AxisName.TailCurlRetracting].arrTargetPoint[1]+1) OR
    	  arrAxisCtrl[AxiseNo.AxisName.TailCurlWhirling].Cmd.arrbRealPoint[1]  ) 
 AND  ( (  arrAxisCtrl[P3AxisNo.P3M1_ColdpreWhirling].Cmd.arrbRealPoint[1] OR arrAxisCtrl[P3AxisNo.P3M1_ColdpreWhirling].Cmd.arrbRealPoint[5] OR arrAxisCtrl[P3AxisNo.P3M1_ColdpreWhirling].Cmd.arrbRealPoint[6] ) OR
                    arrAxisCtrl[P3AxisNo.P3M1_ColdpreRetracting].Cmd.arrbRealPoint[1] )
 OR Mach_Control.TJ_b.AxisConditionEN THEN
	arrAxisCtrl[AxiseNo.AxisName.GluingWhirling].Cmd.GoPoint_Condition[3]:=TRUE;
ELSE
	arrAxisCtrl[AxiseNo.AxisName.GluingWhirling].Cmd.GoPoint_Condition[3]:=FALSE;	
END_IF

IF  Mach_Control.U.WJ_iMode=3 AND arrAxisCtrl[AxiseNo.AxisName.GluingWhirling].Status.Homed  AND arrAxisCtrl[AxiseNo.AxisName.GluingRetracting].Cmd.arrbRealPoint[1] 
AND  ((arrAxisCtrl[AxiseNo.AxisName.TailCurlLine].Status.fSetPos>=arrAxisPar[AxiseNo.AxisName.TailCurlLine].arrTargetPoint[1]-1 AND  arrAxisCtrl[AxiseNo.AxisName.TailCurlRetracting].Status.fSetPos<=arrAxisPar[AxiseNo.AxisName.TailCurlRetracting].arrTargetPoint[1]+1) OR
    	  arrAxisCtrl[AxiseNo.AxisName.TailCurlWhirling].Cmd.arrbRealPoint[1]  ) 
 AND  ( (  arrAxisCtrl[P3AxisNo.P3M1_ColdpreWhirling].Cmd.arrbRealPoint[1] OR arrAxisCtrl[P3AxisNo.P3M1_ColdpreWhirling].Cmd.arrbRealPoint[5] OR arrAxisCtrl[P3AxisNo.P3M1_ColdpreWhirling].Cmd.arrbRealPoint[6] ) OR
                    arrAxisCtrl[P3AxisNo.P3M1_ColdpreRetracting].Cmd.arrbRealPoint[1] )
 OR Mach_Control.TJ_b.AxisConditionEN THEN
	arrAxisCtrl[AxiseNo.AxisName.GluingWhirling].Cmd.GoPoint_Condition[4]:=TRUE;
ELSE
	arrAxisCtrl[AxiseNo.AxisName.GluingWhirling].Cmd.GoPoint_Condition[4]:=FALSE;	
END_IF

IF  Mach_Control.U.WJ_iMode=3 AND arrAxisCtrl[AxiseNo.AxisName.GluingWhirling].Status.Homed  AND arrAxisCtrl[AxiseNo.AxisName.GluingRetracting].Cmd.arrbRealPoint[1] 
AND  ((arrAxisCtrl[AxiseNo.AxisName.TailCurlLine].Status.fSetPos>=arrAxisPar[AxiseNo.AxisName.TailCurlLine].arrTargetPoint[1]-1 AND  arrAxisCtrl[AxiseNo.AxisName.TailCurlRetracting].Status.fSetPos<=arrAxisPar[AxiseNo.AxisName.TailCurlRetracting].arrTargetPoint[1]+1) OR
    	  arrAxisCtrl[AxiseNo.AxisName.TailCurlWhirling].Cmd.arrbRealPoint[1]  ) 
 AND  ( (  arrAxisCtrl[P3AxisNo.P3M1_ColdpreWhirling].Cmd.arrbRealPoint[1] OR arrAxisCtrl[P3AxisNo.P3M1_ColdpreWhirling].Cmd.arrbRealPoint[5] OR arrAxisCtrl[P3AxisNo.P3M1_ColdpreWhirling].Cmd.arrbRealPoint[6] ) OR
                    arrAxisCtrl[P3AxisNo.P3M1_ColdpreRetracting].Cmd.arrbRealPoint[1] )
 OR Mach_Control.TJ_b.AxisConditionEN THEN
	arrAxisCtrl[AxiseNo.AxisName.GluingWhirling].Cmd.GoPoint_Condition[5]:=TRUE;
ELSE
	arrAxisCtrl[AxiseNo.AxisName.GluingWhirling].Cmd.GoPoint_Condition[5]:=FALSE;	
END_IF

IF  Mach_Control.U.WJ_iMode=3 AND arrAxisCtrl[AxiseNo.AxisName.GluingWhirling].Status.Homed  AND arrAxisCtrl[AxiseNo.AxisName.GluingRetracting].Cmd.arrbRealPoint[1] 
AND  ((arrAxisCtrl[AxiseNo.AxisName.TailCurlLine].Status.fSetPos>=arrAxisPar[AxiseNo.AxisName.TailCurlLine].arrTargetPoint[1]-1 AND  arrAxisCtrl[AxiseNo.AxisName.TailCurlRetracting].Status.fSetPos<=arrAxisPar[AxiseNo.AxisName.TailCurlRetracting].arrTargetPoint[1]+1) OR
    	  arrAxisCtrl[AxiseNo.AxisName.TailCurlWhirling].Cmd.arrbRealPoint[1]  ) 
 AND  ( (  arrAxisCtrl[P3AxisNo.P3M1_ColdpreWhirling].Cmd.arrbRealPoint[1] OR arrAxisCtrl[P3AxisNo.P3M1_ColdpreWhirling].Cmd.arrbRealPoint[5] OR arrAxisCtrl[P3AxisNo.P3M1_ColdpreWhirling].Cmd.arrbRealPoint[6] ) OR
                    arrAxisCtrl[P3AxisNo.P3M1_ColdpreRetracting].Cmd.arrbRealPoint[1] )
 OR Mach_Control.TJ_b.AxisConditionEN THEN
	arrAxisCtrl[AxiseNo.AxisName.GluingWhirling].Cmd.GoPoint_Condition[6]:=TRUE;
ELSE
	arrAxisCtrl[AxiseNo.AxisName.GluingWhirling].Cmd.GoPoint_Condition[6]:=FALSE;	
END_IF
*)









//侧贴胶进退
IF  Mach_Control.U.WJ_iMode=3   
 OR Mach_Control.TJ_b.AxisConditionEN THEN
	arrAxisCtrl[AxiseNo.AxisName.GluingRetracting].Cmd.Home_Condition:=TRUE;
ELSE
	arrAxisCtrl[AxiseNo.AxisName.GluingRetracting].Cmd.Home_Condition:=FALSE;	
END_IF

IF  Mach_Control.U.WJ_iMode=3 AND arrAxisCtrl[AxiseNo.AxisName.GluingRetracting].Status.Homed AND arrAxisCtrl[AxiseNo.AxisName.GluingUpDown].Cmd.arrbRealPoint[9]  
 OR Mach_Control.TJ_b.AxisConditionEN THEN
	arrAxisCtrl[AxiseNo.AxisName.GluingRetracting].Cmd.GoPoint_Condition[1]:=TRUE;
ELSE
	arrAxisCtrl[AxiseNo.AxisName.GluingRetracting].Cmd.GoPoint_Condition[1]:=FALSE;	
END_IF

IF  Mach_Control.U.WJ_iMode=3 AND arrAxisCtrl[AxiseNo.AxisName.GluingRetracting].Status.Homed AND arrAxisCtrl[AxiseNo.AxisName.GluingUpDown].Cmd.arrbRealPoint[9]
AND arrAxisCtrl[AxiseNo.AxisName.GluingWhirling].Cmd.arrbRealPoint[1] AND arrCyCtrl[arrCyNo.CylinderName.GlueClampsCy].Status.OFFState
 OR Mach_Control.TJ_b.AxisConditionEN THEN
	arrAxisCtrl[AxiseNo.AxisName.GluingRetracting].Cmd.GoPoint_Condition[2]:=TRUE;
ELSE
	arrAxisCtrl[AxiseNo.AxisName.GluingRetracting].Cmd.GoPoint_Condition[2]:=FALSE;	
END_IF

IF  Mach_Control.U.WJ_iMode=3 AND arrAxisCtrl[AxiseNo.AxisName.GluingRetracting].Status.Homed AND arrAxisCtrl[AxiseNo.AxisName.GluingUpDown].Cmd.arrbRealPoint[9]
AND arrAxisCtrl[AxiseNo.AxisName.GluingWhirling].Cmd.arrbRealPoint[2]AND arrCyCtrl[arrCyNo.CylinderName.GlueClampsCy].Status.OFFState
 OR Mach_Control.TJ_b.AxisConditionEN THEN
	arrAxisCtrl[AxiseNo.AxisName.GluingRetracting].Cmd.GoPoint_Condition[3]:=TRUE;
ELSE
	arrAxisCtrl[AxiseNo.AxisName.GluingRetracting].Cmd.GoPoint_Condition[3]:=FALSE;	
END_IF

IF  Mach_Control.U.WJ_iMode=3 AND arrAxisCtrl[AxiseNo.AxisName.GluingRetracting].Status.Homed AND arrAxisCtrl[AxiseNo.AxisName.GluingUpDown].Cmd.arrbRealPoint[9]
AND arrAxisCtrl[AxiseNo.AxisName.GluingWhirling].Cmd.arrbRealPoint[3]
 OR Mach_Control.TJ_b.AxisConditionEN THEN
	arrAxisCtrl[AxiseNo.AxisName.GluingRetracting].Cmd.GoPoint_Condition[4]:=TRUE;
ELSE
	arrAxisCtrl[AxiseNo.AxisName.GluingRetracting].Cmd.GoPoint_Condition[4]:=FALSE;	
END_IF

IF  Mach_Control.U.WJ_iMode=3 AND arrAxisCtrl[AxiseNo.AxisName.GluingRetracting].Status.Homed AND arrAxisCtrl[AxiseNo.AxisName.GluingUpDown].Cmd.arrbRealPoint[9]
AND arrAxisCtrl[AxiseNo.AxisName.GluingWhirling].Cmd.arrbRealPoint[4]
 OR Mach_Control.TJ_b.AxisConditionEN THEN
	arrAxisCtrl[AxiseNo.AxisName.GluingRetracting].Cmd.GoPoint_Condition[5]:=TRUE;
ELSE
	arrAxisCtrl[AxiseNo.AxisName.GluingRetracting].Cmd.GoPoint_Condition[5]:=FALSE;	
END_IF


IF  Mach_Control.U.WJ_iMode=3 AND arrAxisCtrl[AxiseNo.AxisName.GluingRetracting].Status.Homed AND arrAxisCtrl[AxiseNo.AxisName.GluingUpDown].Cmd.arrbRealPoint[9] 
 OR Mach_Control.TJ_b.AxisConditionEN THEN
	arrAxisCtrl[AxiseNo.AxisName.GluingRetracting].Cmd.GoPoint_Condition[6]:=TRUE;
ELSE
	arrAxisCtrl[AxiseNo.AxisName.GluingRetracting].Cmd.GoPoint_Condition[6]:=FALSE;	
END_IF


//侧贴胶升降
IF  Mach_Control.U.WJ_iMode=3   
 OR Mach_Control.TJ_b.AxisConditionEN THEN
	arrAxisCtrl[AxiseNo.AxisName.GluingUpDown].Cmd.Home_Condition:=TRUE;
ELSE
	arrAxisCtrl[AxiseNo.AxisName.GluingUpDown].Cmd.Home_Condition:=FALSE;	
END_IF

IF  Mach_Control.U.WJ_iMode=3 AND arrAxisCtrl[AxiseNo.AxisName.GluingUpDown].Status.Homed   
 OR Mach_Control.TJ_b.AxisConditionEN THEN
	arrAxisCtrl[AxiseNo.AxisName.GluingUpDown].Cmd.GoPoint_Condition[1]:=TRUE;
ELSE
	arrAxisCtrl[AxiseNo.AxisName.GluingUpDown].Cmd.GoPoint_Condition[1]:=FALSE;	
END_IF

IF  Mach_Control.U.WJ_iMode=3 AND arrAxisCtrl[AxiseNo.AxisName.GluingUpDown].Status.Homed AND arrAxisCtrl[AxiseNo.AxisName.GluingRetracting].Cmd.arrbRealPoint[1]  
 OR Mach_Control.TJ_b.AxisConditionEN THEN
	arrAxisCtrl[AxiseNo.AxisName.GluingUpDown].Cmd.GoPoint_Condition[2]:=TRUE;
ELSE
	arrAxisCtrl[AxiseNo.AxisName.GluingUpDown].Cmd.GoPoint_Condition[2]:=FALSE;	
END_IF

IF  Mach_Control.U.WJ_iMode=3 AND arrAxisCtrl[AxiseNo.AxisName.GluingUpDown].Status.Homed AND arrAxisCtrl[AxiseNo.AxisName.GluingRetracting].Cmd.arrbRealPoint[1]  
 OR Mach_Control.TJ_b.AxisConditionEN THEN
	arrAxisCtrl[AxiseNo.AxisName.GluingUpDown].Cmd.GoPoint_Condition[3]:=TRUE;
ELSE
	arrAxisCtrl[AxiseNo.AxisName.GluingUpDown].Cmd.GoPoint_Condition[3]:=FALSE;	
END_IF


IF  Mach_Control.U.WJ_iMode=3 AND arrAxisCtrl[AxiseNo.AxisName.GluingUpDown].Status.Homed AND arrAxisCtrl[AxiseNo.AxisName.GluingRetracting].Cmd.arrbRealPoint[1]  
 OR Mach_Control.TJ_b.AxisConditionEN THEN
	arrAxisCtrl[AxiseNo.AxisName.GluingUpDown].Cmd.GoPoint_Condition[4]:=TRUE;
ELSE
	arrAxisCtrl[AxiseNo.AxisName.GluingUpDown].Cmd.GoPoint_Condition[4]:=FALSE;	
END_IF



IF  Mach_Control.U.WJ_iMode=3 AND arrAxisCtrl[AxiseNo.AxisName.GluingUpDown].Status.Homed AND arrAxisCtrl[AxiseNo.AxisName.GluingRetracting].Cmd.arrbRealPoint[1]  
 OR Mach_Control.TJ_b.AxisConditionEN THEN
	arrAxisCtrl[AxiseNo.AxisName.GluingUpDown].Cmd.GoPoint_Condition[5]:=TRUE;
ELSE
	arrAxisCtrl[AxiseNo.AxisName.GluingUpDown].Cmd.GoPoint_Condition[5]:=FALSE;	
END_IF


IF  Mach_Control.U.WJ_iMode=3 AND arrAxisCtrl[AxiseNo.AxisName.GluingUpDown].Status.Homed AND arrAxisCtrl[AxiseNo.AxisName.GluingRetracting].Cmd.arrbRealPoint[1]  
 OR Mach_Control.TJ_b.AxisConditionEN THEN
	arrAxisCtrl[AxiseNo.AxisName.GluingUpDown].Cmd.GoPoint_Condition[6]:=TRUE;
ELSE
	arrAxisCtrl[AxiseNo.AxisName.GluingUpDown].Cmd.GoPoint_Condition[6]:=FALSE;	
END_IF


IF  Mach_Control.U.WJ_iMode=3 AND arrAxisCtrl[AxiseNo.AxisName.GluingUpDown].Status.Homed AND arrAxisCtrl[AxiseNo.AxisName.GluingRetracting].Cmd.arrbRealPoint[1]  
 OR Mach_Control.TJ_b.AxisConditionEN THEN
	arrAxisCtrl[AxiseNo.AxisName.GluingUpDown].Cmd.GoPoint_Condition[7]:=TRUE;
ELSE
	arrAxisCtrl[AxiseNo.AxisName.GluingUpDown].Cmd.GoPoint_Condition[7]:=FALSE;	
END_IF

IF  Mach_Control.U.WJ_iMode=3 AND arrAxisCtrl[AxiseNo.AxisName.GluingUpDown].Status.Homed AND arrAxisCtrl[AxiseNo.AxisName.GluingRetracting].Cmd.arrbRealPoint[1]  
 OR Mach_Control.TJ_b.AxisConditionEN THEN
	arrAxisCtrl[AxiseNo.AxisName.GluingUpDown].Cmd.GoPoint_Condition[8]:=TRUE;
ELSE
	arrAxisCtrl[AxiseNo.AxisName.GluingUpDown].Cmd.GoPoint_Condition[8]:=FALSE;	
END_IF
IF  Mach_Control.U.WJ_iMode=3 AND arrAxisCtrl[AxiseNo.AxisName.GluingUpDown].Status.Homed AND arrAxisCtrl[AxiseNo.AxisName.GluingRetracting].Cmd.arrbRealPoint[1]  
 OR Mach_Control.TJ_b.AxisConditionEN THEN
	arrAxisCtrl[AxiseNo.AxisName.GluingUpDown].Cmd.GoPoint_Condition[9]:=TRUE;
ELSE
	arrAxisCtrl[AxiseNo.AxisName.GluingUpDown].Cmd.GoPoint_Condition[9]:=FALSE;	
END_IF
END_ACTION

ACTION Sticker_Alarm:

TJ_AlarmTon[1](IN:= , PT:=T#300MS , Q=> , ET=> );//
//TJ_AlarmTon[2](IN:= , PT:=T#300MS , Q=> , ET=> );//
TJ_AlarmTon[3](IN:= , PT:=T#300MS , Q=> , ET=> );//
//TJ_AlarmTon[4](IN:= , PT:=T#300MS , Q=> , ET=> );//
TJ_AlarmTon[5](IN:= , PT:=T#100MS , Q=> , ET=> );//
TJ_AlarmTon[6](IN:= , PT:=T#50MS , Q=> , ET=> );//
TJ_AlarmTon[7](IN:= , PT:=T#1000MS , Q=> , ET=> );//

IF  arrCyCtrl[arrCyNo.ElectValveName.BlueGlueVacuum1].Io.DOStatus1 AND NOT arrCyCtrl[arrCyNo.ElectValveName.BlueGlueVacuum1].Io.DIOnSwitch THEN
	IF NOT TJ_AlarmTon[1].Q  THEN
		TJ_AlarmTon[1].IN:=TRUE;
	ELSE
			Mach_Control.TJ_b.Error[1] :=TRUE;//备胶组件蓝胶真空1报警
	END_IF
ELSE
		TJ_AlarmTon[1].IN:=FALSE;
END_IF
(*
IF  arrCyCtrl[arrCyNo.ElectValveName.BlueGlueVacuum2].Cmd.bON AND NOT arrCyCtrl[arrCyNo.ElectValveName.BlueGlueVacuum2].Io.DIOnSwitch THEN
	IF NOT TJ_AlarmTon[2].Q THEN
		TJ_AlarmTon[2].IN:=TRUE;
	ELSE
			;//Mach_Control.TJ_b.Error[2] :=TRUE;//备胶组件蓝胶真空2报警
	END_IF
ELSE
		TJ_AlarmTon[2].IN:=FALSE;
END_IF*)

IF  arrCyCtrl[arrCyNo.ElectValveName.codeGlueVacuum1].Io.DOStatus1  AND NOT arrCyCtrl[arrCyNo.ElectValveName.codeGlueVacuum1].Io.DIOnSwitch THEN
	IF NOT TJ_AlarmTon[3].Q THEN
		TJ_AlarmTon[3].IN:=TRUE;
	ELSE
			Mach_Control.TJ_b.Error[3] :=TRUE;//备胶组件二维码真空1报警
			Mach_Control.TJ_b.Scan_Men[1].Scan_gross:=0;
			Mach_Control.TJ_b.Scan_Men[2].Scan_gross:=0;
			Mach_Control.TJ_b.Scan_Men[3].Scan_gross:=0;
	END_IF
ELSE
		TJ_AlarmTon[3].IN:=FALSE;
END_IF

(*
IF  arrCyCtrl[arrCyNo.ElectValveName.codeGlueVacuum2].Cmd.bON  AND NOT arrCyCtrl[arrCyNo.ElectValveName.codeGlueVacuum2].Io.DIOnSwitch THEN
	IF NOT TJ_AlarmTon[4].Q THEN
		TJ_AlarmTon[4].IN:=TRUE;
	ELSE
			;//Mach_Control.TJ_b.Error[4] :=TRUE;//备胶组件二维码真空2报警
	END_IF
ELSE
		TJ_AlarmTon[4].IN:=FALSE;
END_IF
*)

IF  arrCyCtrl[arrCyNo.ElectValveName.PastesGlueVacuum].Io.DOStatus1  AND NOT arrCyCtrl[arrCyNo.ElectValveName.PastesGlueVacuum].Io.DIOnSwitch  
	AND NOT (Sticker_Step2>=400 )THEN
	IF NOT TJ_AlarmTon[5].Q THEN
		TJ_AlarmTon[5].IN:=TRUE;
	ELSE
			Mach_Control.TJ_b.Error[5] :=TRUE;//备胶组件贴胶胶头真空报警
			arrCyCtrl[arrCyNo.ElectValveName.PastesGlueVacuum].Cmd.bOFF:=TRUE;
	END_IF
ELSE
		TJ_AlarmTon[5].IN:=FALSE;
END_IF

IF NOT arrCyCtrl[arrCyNo.ElectValveName.PastesGlueVacuum].Io.DOStatus1 AND arrCyCtrl[arrCyNo.ElectValveName.PastesGlueVacuum].Io.DIOnSwitch 
	AND NOT (Sticker_Step2>=400 )THEN
	IF NOT TJ_AlarmTon[7].Q THEN
		TJ_AlarmTon[7].IN:=TRUE;
	ELSE
			Mach_Control.TJ_b.Error[7] :=TRUE;//备胶组件贴胶头没开真空有真空信号报警
			
	END_IF
ELSE
		TJ_AlarmTon[7].IN:=FALSE;
END_IF



IF  Sticker_Step1=9999  THEN
	IF NOT TJ_AlarmTon[6].Q THEN
		TJ_AlarmTon[6].IN:=TRUE;
	ELSE
			Mach_Control.TJ_b.Error[6] :=TRUE;//找不到Mark孔报警
			StandbyCode_Start:=FALSE;
			StandbyBule_Start:=FALSE;
	END_IF
ELSE
		TJ_AlarmTon[6].IN:=FALSE;
END_IF

IF  	Mach_Control.TJ_b.Error[1]//备胶组件蓝胶真空1报警
	OR Mach_Control.TJ_b.Error[2] //备胶组件蓝胶真空2报警
	OR Mach_Control.TJ_b.Error[3] //备胶组件二维码真空1报警
	OR Mach_Control.TJ_b.Error[4] //备胶组件二维码真空2报警
	OR Mach_Control.TJ_b.Error[5] //备胶组件贴胶胶头真空报警
	THEN
	TJ_Error:=TRUE;	
	StandbyCode_Start:=FALSE;
	StandbyBule_Start:=FALSE;
	END_IF

IF (Mach_Control.TJ_b.Error[5] OR Mach_Control.TJ_b.Error[6])  AND fTSticker_AlarmRest.Q THEN	
	Sticker_Step1:=0;
END_IF
(*
IF Mach_Control.TJ_b.Scan_Men[3].Scan_gross<>1 AND NOT Mach_Control.TJ_b.ScanMode THEN
	Mach_Control.TJ_b.Scan_TS:=TRUE;
	ELSE
	Mach_Control.TJ_b.Scan_TS:=FALSE;
END_IF

*)
//贴胶报警复位处理
rSticker_AlarmRest(CLK:=Sys_Control.btn.System_Rrestbtn , Q=> );
fTSticker_AlarmRest(CLK:=Sys_Control.btn.System_Rrestbtn , Q=> );
IF Mach_Control.U.TJ_iMode=3 THEN//在手动状态下，复位报警
		IF fTSticker_AlarmRest.Q THEN
				MEMSET(ADR(Mach_Control.TJ_b.Error),0,SIZEOF(Mach_Control.TJ_b.Error)); // 贴胶报警复位
				TJ_Error:=FALSE;
				
		END_IF
END_IF
Mach_Control.TJ_b.Error[9];//贴胶治具有信号无记忆报警
Mach_Control.TJ_b.Error[11];//叠台贴胶头贴胶时无贴胶报警
END_ACTION

ACTION Sticker_Gohome:
StickerGohome_TON[1](PT:=T#1S);
StickerGohome_TON[2](PT:=T#1S);
StickerGohome_TON[3](PT:=T#1S);
StickerGohome_TON[4](PT:=T#1S);
StickerGohome_TON[5](PT:=T#1S);
StickerGohome_TON[6](PT:=T#1S);
StickerGohome_TON[7](PT:=T#1S);
Sticker_GohomeOverTon(IN:= , PT:=T#120S , Q=> , ET=> );//贴胶回原点超时报警延时

//判断贴胶回原点是否完成
IF arrAxisCtrl[AxiseNo.AxisName.GluingRetracting].Status.Homed AND arrAxisCtrl[AxiseNo.AxisName.GluingRetracting].Status.NoMoving  AND 
	arrAxisCtrl[AxiseNo.AxisName.GluingUpDown].Status.Homed AND arrAxisCtrl[AxiseNo.AxisName.GluingUpDown].Status.NoMoving   AND
	arrAxisCtrl[AxiseNo.AxisName.GluingLine].Status.Homed AND arrAxisCtrl[AxiseNo.AxisName.GluingLine].Status.NoMoving AND
	arrAxisCtrl[AxiseNo.AxisName.GluingWhirling].Status.Homed AND arrAxisCtrl[AxiseNo.AxisName.GluingWhirling].Status.NoMoving  AND TJIniti_Done THEN	 
		Mach_Control.TJ_b.TJIniti_Done:=TRUE;//复位贴胶初始化完成	
ELSE
		Mach_Control.TJ_b.TJIniti_Done:=FALSE;//复位贴胶初始化完成		
END_IF


IF Mach_Control.U.WJ_iMode=3 THEN//在手动状态下
		IF r_Sticker_init.Q THEN
			StickerStep0:=0;
			TJIniti_Done:=FALSE;
		END_IF	
END_IF		
IF Sticker_GohomeOverTon.Q THEN
	Sticker_GohomeOverTon.IN:=FALSE;
	StickerStep0:=0;
	Mach_Control.TJ_b.Error[8]:=TRUE; //贴胶回原超时报警
END_IF


r_Sticker_init(CLK:=Mach_Control.TJ_b.TJIniti_Hbtn(* OR Mach_Control.DT_b.ALLIniti_Hbtn *), Q=> );
f_Sticker_init(CLK:=Mach_Control.TJ_b.TJIniti_Hbtn (*OR Mach_Control.DT_b.ALLIniti_Hbtn *), Q=> );
tStickerTON(IN:= , PT:= , Q=> , ET=> );
IF Mach_Control.U.WJ_iMode=3 THEN//在手动状态下
	CASE StickerStep0 OF
		0://
			IF f_Sticker_init.Q THEN		
				StickerStep0:=1;
				Sticker_Step0:=0;
				Sticker_Step1:=0;
				Sticker_Step2:=0;		
				CellMemory[Mach_Control.TJ_b.TJ_Memory].Cell:=FALSE;
				Sticker_GohomeOverTon.IN:=TRUE;
			END_IF
		1:
				Mach_Control.TJ_b.StickPermit:=FALSE;//贴胶允许
				Mach_Control.TJ_b.StickFinish:=FALSE;//贴胶完成	
				Mach_Control.TJ_b.StickMark_L1 :=FALSE;//左短边1贴胶完成
				Mach_Control.TJ_b.StickMark_L2 :=FALSE;//左短边2贴胶完成
				Mach_Control.TJ_b.StickMark_R1 :=FALSE;//右短边1贴胶完成
				Mach_Control.TJ_b.StickMark_R2 :=FALSE;//右短边2贴胶完成		
				Mach_Control.TJ_b.StickMark1_L :=FALSE;//右短边2贴胶完成		
				Mach_Control.TJ_b.StickMark1_L2 :=FALSE;//右短边2贴胶完成		
				Mach_Control.TJ_b.Sticking_L:=FALSE;//左短边贴胶
				Mach_Control.TJ_b.Sticking_R:=FALSE;//右短边贴胶
				Mach_Control.TJ_b.Sticking_Lg:=FALSE;//非极耳侧长边贴胶
				Mach_Control.TJ_b.Sticking_Lg2:=FALSE;//极耳侧长边贴胶				
				TJIniti_Done:=FALSE;//复位贴胶初始化完成	
				Mach_Control.TJ_b.StickerFlag:=FALSE;
				Mach_Control.TJ_b.StickerDone:=FALSE;
				Mach_Control.TJ_b.StickerOffloadingDone:=FALSE;	
				IF NOT TJIniti_Done THEN
					StickerStep0:=10;
				END_IF
		10://贴胶冶具气缸开， 贴胶NG气缸回
			arrCyCtrl[arrCyNo.CylinderName.PullGlueModelCy].Cmd.bON:=TRUE;//贴胶冶具夹爪张开
			arrCyCtrl[arrCyNo.CylinderName.GlueNGCy].Cmd.bOFF:=TRUE;//贴胶NG回
			IF arrCyCtrl[arrCyNo.CylinderName.PullGlueModelCy].Io.DIONSwitch AND arrCyCtrl[arrCyNo.CylinderName.GlueNGCy].Io.DIOFFSwitch THEN
				StickerStep0:=20;
			END_IF
		20://贴胶头进退回原
			arrAxisCtrl[AxiseNo.AxisName.GluingRetracting].Cmd.bHome:=TRUE;//贴胶头进退轴回原点
			StickerStep0:=25;					
		25://判断帖胶头进退轴回原点是否完成	
			StickerGohome_TON[1].IN:=TRUE;
		IF arrAxisCtrl[AxiseNo.AxisName.GluingRetracting].Status.Homed AND arrAxisCtrl[AxiseNo.AxisName.GluingRetracting].Status.NoMoving  AND StickerGohome_TON[1].Q THEN
			arrAxisCtrl[AxiseNo.AxisName.GluingRetracting].Cmd.bHome:=FALSE;
			StickerGohome_TON[1].IN:=FALSE;
			StickerStep0:=30;
		END_IF				
		30://贴胶头平移轴移动至初始位
			IF  arrAxisCtrl[AxiseNo.AxisName.GluingRetracting].Status.Homed AND arrAxisCtrl[AxiseNo.AxisName.GluingRetracting].Status.NoMoving THEN
					IF arrAxisCtrl[AxiseNo.AxisName.GluingRetracting].Cmd.arrbRealPoint[1] AND  arrAxisCtrl[AxiseNo.AxisName.GluingRetracting].Status.NoMoving  THEN
						arrAxisCtrl[AxiseNo.AxisName.GluingRetracting].Cmd.iGoSetPos:=0;
						StickerStep0:=40;	
					ELSE
						arrAxisCtrl[AxiseNo.AxisName.GluingRetracting].Cmd.iGoSetPos:=1;//贴胶头进退去初始位
					END_IF
			END_IF			
		40://切胶气缸伸出，拉胶气缸伸出，拉胶升降轴回原点
				arrCyCtrl[arrCyNo.CylinderName.codeGlueCutCy].Cmd.bON:=TRUE;//贴胶切二维码胶气缸伸出
				arrCyCtrl[arrCyNo.CylinderName.GlueCutCy].Cmd.bON:=TRUE;//贴胶切胶气缸伸出
				arrCyCtrl[arrCyNo.CylinderName.PullGlueCy].Cmd.bON:=TRUE;//拉胶气缸伸出
				IF	arrCyCtrl[arrCyNo.CylinderName.codeGlueCutCy].Io.DIOnSwitch 
				AND arrCyCtrl[arrCyNo.CylinderName.GlueCutCy].Io.DIOnSwitch 
				AND arrCyCtrl[arrCyNo.CylinderName.PullGlueCy].Io.DIOnSwitch THEN
					StickerStep0:=50;	
				END_IF
		50:		
				arrAxisCtrl[AxiseNo.AxisName.GluingUpDown].Cmd.bHome:=TRUE;//拉胶升降轴回原点		
				StickerStep0:=53;
		53:	//判断拉胶升降轴回原点是否完成	
					StickerGohome_TON[2].IN:=TRUE;
				IF arrAxisCtrl[AxiseNo.AxisName.GluingUpDown].Status.Homed AND arrAxisCtrl[AxiseNo.AxisName.GluingUpDown].Status.NoMoving  AND StickerGohome_TON[2].Q THEN
					arrAxisCtrl[AxiseNo.AxisName.GluingUpDown].Cmd.bHome:=FALSE;//拉胶升降轴回原点
					StickerGohome_TON[2].IN:=FALSE;
					StickerStep0:=55;
				END_IF			
		55://拉胶升降轴去踢废避让位
				IF  arrAxisCtrl[AxiseNo.AxisName.GluingUpDown].Status.Homed AND arrAxisCtrl[AxiseNo.AxisName.GluingUpDown].Status.NoMoving THEN
						IF arrAxisCtrl[AxiseNo.AxisName.GluingUpDown].Cmd.arrbRealPoint[9]  AND  arrAxisCtrl[AxiseNo.AxisName.GluingUpDown].Status.NoMoving THEN
							arrAxisCtrl[AxiseNo.AxisName.GluingUpDown].Cmd.iGoSetPos:=0;
							StickerStep0:=60;	
						ELSE
							arrAxisCtrl[AxiseNo.AxisName.GluingUpDown].Cmd.iGoSetPos:=9;//拉胶升降轴至踢废胶避让位
						END_IF
				END_IF				
		60://贴胶夹电芯气缸张开，侧贴胶平移轴回原点
				arrCyCtrl[arrCyNo.CylinderName.GlueClampsCy].Cmd.bOFF:=TRUE;//贴胶夹爪气缸张开
				IF 	arrCyCtrl[arrCyNo.CylinderName.GlueClampsCy].Io.DIOFFSwitch AND
                  GluingLineagree THEN		
					arrAxisCtrl[AxiseNo.AxisName.GluingLine].Cmd.bHome:=TRUE;//侧贴胶平移回原
					StickerStep0:=65;	
				ELSE	
					Mach_Control.TJ_b.Error[10]:=TRUE; //侧贴胶平移回原点时条件不满足报警
					StickerStep0:=0;	
				END_IF			
		65://判断侧贴胶平移是否回原完成
				StickerGohome_TON[3].IN:=TRUE;
				IF arrAxisCtrl[AxiseNo.AxisName.GluingLine].Status.Homed AND arrAxisCtrl[AxiseNo.AxisName.GluingLine].Status.NoMoving  AND StickerGohome_TON[3].Q THEN
					arrAxisCtrl[AxiseNo.AxisName.GluingLine].Cmd.bHome:=FALSE;
					StickerGohome_TON[3].IN:=FALSE;
					StickerStep0:=70;
				END_IF
		70://侧贴胶平移移动至左短边侧贴胶位1
			IF  arrAxisCtrl[AxiseNo.AxisName.GluingLine].Status.Homed AND arrAxisCtrl[AxiseNo.AxisName.GluingLine].Status.NoMoving THEN
					IF arrAxisCtrl[AxiseNo.AxisName.GluingLine].Cmd.arrbRealPoint[1] THEN
						arrAxisCtrl[AxiseNo.AxisName.GluingLine].Cmd.iGoSetPos:=0;
						StickerStep0:=80;	
					ELSE
						arrAxisCtrl[AxiseNo.AxisName.GluingLine].Cmd.iGoSetPos:=1;//
					END_IF
			END_IF			
		80://贴胶夹电芯气缸张开，侧贴胶旋转回原点
				arrCyCtrl[arrCyNo.CylinderName.GlueClampsCy].Cmd.bOFF:=TRUE;//贴胶夹爪气缸张开
				IF 	arrCyCtrl[arrCyNo.CylinderName.GlueClampsCy].Io.DIOFFSwitch AND
                    Mach_Control.TJ_b.WhirlingSafe THEN
					arrAxisCtrl[AxiseNo.AxisName.GluingWhirling].Cmd.bHome:=TRUE;//侧贴胶旋转轴回原点
					StickerStep0:=85;
				END_IF		
		85://判断侧贴胶旋转回原是否完成
				StickerGohome_TON[4].IN:=TRUE;
				IF arrAxisCtrl[AxiseNo.AxisName.GluingWhirling].Status.Homed AND arrAxisCtrl[AxiseNo.AxisName.GluingWhirling].Status.NoMoving  AND StickerGohome_TON[4].Q THEN
					StickerStep0:=90;
					arrAxisCtrl[AxiseNo.AxisName.GluingWhirling].Cmd.bHome:=FALSE;//侧贴胶旋转轴回原点
					StickerGohome_TON[4].IN:=FALSE;
				END_IF
		90://侧贴胶旋转去上电芯位
			IF  arrAxisCtrl[AxiseNo.AxisName.GluingWhirling].Status.Homed AND arrAxisCtrl[AxiseNo.AxisName.GluingWhirling].Status.NoMoving THEN
					IF arrAxisCtrl[AxiseNo.AxisName.GluingWhirling].Cmd.arrbRealPoint[5] AND arrAxisCtrl[AxiseNo.AxisName.GluingWhirling].Status.NoMoving THEN
						arrAxisCtrl[AxiseNo.AxisName.GluingWhirling].Cmd.iGoSetPos:=0;
						StickerStep0:=110;	
					ELSE
						arrAxisCtrl[AxiseNo.AxisName.GluingWhirling].Cmd.iGoSetPos:=5;//旋转至上电芯位
					END_IF
			END_IF	
		110://判断侧贴胶平移轴回原点是否完成，侧贴胶旋转轴回原点是否完成
			IF arrAxisCtrl[AxiseNo.AxisName.GluingLine].Status.Homed AND arrAxisCtrl[AxiseNo.AxisName.GluingLine].Status.NoMoving AND 
				arrAxisCtrl[AxiseNo.AxisName.GluingWhirling].Status.Homed AND arrAxisCtrl[AxiseNo.AxisName.GluingWhirling].Status.NoMoving 
			THEN
				Sticker_GohomeOverTon.IN:=FALSE;
				TJIniti_Done:=TRUE;
				StickerStep0:=0;
			END_IF
	END_CASE			
END_IF
END_ACTION

ACTION StickGlue_Init:
		arrCyCtrl[arrCyNo.CylinderName.codeGlueCutCy].Cmd.bON:=TRUE;//切二维胶伸出
		arrCyCtrl[arrCyNo.CylinderName.CodeGluePressCy].Cmd.bOFF:=TRUE;//压二维码胶收回
		arrCyCtrl[arrCyNo.CylinderName.CodeStandbyGlueCy].Cmd.bOFF:=TRUE;//备二维码胶收回		
		arrCyCtrl[arrCyNo.CylinderName.GlueCutCy].Cmd.bON:=TRUE;//切胶伸出
		arrCyCtrl[arrCyNo.CylinderName.GluePressCy].Cmd.bOFF:=TRUE;//压胶气缸收回
		arrCyCtrl[arrCyNo.CylinderName.StandbyGlueCy].Cmd.bOFF:=TRUE;//备胶气缸收回	
		arrCyCtrl[arrCyNo.CylinderName.PullGlueCy].Cmd.bON:=TRUE;//贴胶拉胶气缸伸出
		arrCyCtrl[arrCyNo.CylinderName.PullGlueCy].Cmd.bOFF:=TRUE;//贴胶冶具气缸收回
		arrCyCtrl[arrCyNo.CylinderName.PullGlueCy].Cmd.bOFF:=TRUE;//贴胶冶具气缸收回
		arrCyCtrl[arrCyNo.CylinderName.PullGluePoleCy].Cmd.bOFF:=TRUE;//拉胶锁紧气缸收回	
		arrCyCtrl[arrCyNo.CylinderName.GlueNGCy].Cmd.bOFF:=TRUE;//踢废胶收回		
		arrCyCtrl[arrCyNo.CylinderName.GlueClampsCy].Cmd.bON:=TRUE;//贴胶夹爪气缸张开
END_ACTION

ACTION TailCurl_Alarm:
//尾卷报警复位处理
rTailCurl_AlarmRest(CLK:=Sys_Control.btn.System_Rrestbtn , Q=> );
fTailCurl_AlarmRest(CLK:=Sys_Control.btn.System_Rrestbtn , Q=> );
IF Mach_Control.U.WJ_iMode=3 THEN//在手动状态下，复位报警
		IF fTailCurl_AlarmRest.Q THEN
				MEMSET(ADR(Mach_Control.WJ_b.Error),0,SIZEOF(Mach_Control.WJ_b.Error)); // 叠台报警复位
		END_IF
END_IF


   IF arrAxisPar[AxiseNo.AxisName.TailCurlSEPTALine].arrTargetPoint[3]=0 THEN 
	   arrAxisPar[AxiseNo.AxisName.TailCurlSEPTALine].arrTargetPoint[3]:=500 ;	
	END_IF
     
	TailCurlAxisbstop_R(CLK:= arrAxisbstop[AxiseNo.AxisName.TailCurlLine] , Q=> );//HMI轴停止上升沿
    TailCurlAxisbstop_F(CLK:= arrAxisbstop[AxiseNo.AxisName.TailCurlLine] , Q=> );//HMI轴停止下降沿

     IF TailCurlAxisbstop_R.Q AND Mach_Control.U.WJ_iMode=3 THEN 
        arrAxisCtrl[AxiseNo.AxisName.TailCurlLine].Cmd.bStop:=TRUE;
     END_IF
 
     IF TailCurlAxisbstop_F.Q  AND  Mach_Control.U.WJ_iMode=3  THEN 
         arrAxisCtrl[AxiseNo.AxisName.TailCurlLine].Cmd.bStop:=FALSE;
     END_IF
	
    TailCurl_WJJMPY_Xzb:=arrAxisPar[AxiseNo.AxisName.TailCurlSEPTALine].arrTargetPoint[3]+arrAxisCtrl[AxiseNo.AxisName.TailCurlSEPTALine].Status.fActPos;

    IF TailCurlStep3=105 AND NOT arrAxisCtrl[AxiseNo.AxisName.TailCurlSEPTALine].Cmd.arrbRealPoint[2] AND arrAxisCtrl[AxiseNo.AxisName.TailCurlLine].Status.Moving
		 AND (*arrAxisCtrl[AxiseNo.AxisName.TailCurlSEPTALine].Status.Homed  AND*) arrAxisCtrl[AxiseNo.AxisName.TailCurlLine].Status.Homed AND
         ABS( TailCurl_WJJMPY_Xzb-arrAxisCtrl[AxiseNo.AxisName.TailCurlLine].Status.fActPos) <100 THEN
	   Mach_Control.WJ_b.Error[26]:=TRUE;//尾卷夹平移防撞软限位报警
	END_IF
	
	WJError_r(CLK:= Mach_Control.WJ_b.Error[26] , Q=> );
	IF WJError_r.Q THEN 
	  // arrAxisCtrl[AxiseNo.AxisName.TailCurlSEPTALine].Cmd.bStop:=TRUE;
       arrAxisCtrl[AxiseNo.AxisName.TailCurlLine].Cmd.bStop :=TRUE;	
	END_IF
	
    IF  P2M2_sysControl.btn.System_Rrestbtn  THEN
       arrAxisCtrl[AxiseNo.AxisName.TailCurlSEPTALine].Cmd.bStop:=FALSE;
       arrAxisCtrl[AxiseNo.AxisName.TailCurlLine].Cmd.bStop :=FALSE;
	END_IF
	
		IF arrAxisCtrl[AxiseNo.AxisName.SCurlingneedleWhirling].Cmd.arrbRealPoint[1] AND NOT   arrAxisCtrl[AxiseNo.AxisName.SCurlingneedleWhirling].Io.biHomeSwitch AND 
            arrAxisCtrl[AxiseNo.AxisName.SCurlingneedleWhirling].Status.NoMoving  THEN
			 Mach_Control.WJ_b.Error[4]:=TRUE;//短卷针旋转在初始位原点传感器不亮报警
		END_IF
		
		IF arrAxisCtrl[AxiseNo.AxisName.LCurlingneedleWhirling].Cmd.arrbRealPoint[1] AND NOT   arrAxisCtrl[AxiseNo.AxisName.LCurlingneedleWhirling].Io.biHomeSwitch AND  
            arrAxisCtrl[AxiseNo.AxisName.LCurlingneedleWhirling].Status.NoMoving THEN
			 Mach_Control.WJ_b.Error[6]:=TRUE;//长卷针旋转在初始位原点传感器不亮报警
		END_IF

GluebHaveTON(PT:=T#500MS);
GluebHaveTON.IN:=(TailCurlStep3=332 AND Mach_Control.se.GluebHave AND NOT CellMemory[Mach_Control.TJ_b.TJ_Memory].Cell );
IF GluebHaveTON.Q AND arrAxisCtrl[AxiseNo.AxisName.GluingWhirling].Status.NoMoving THEN
	Mach_Control.TJ_b.Error[9]:=TRUE; //贴胶夹爪有信号无记忆报警
	;
END_IF

IF Par.stWJ_date.Hotcount>=Par.stWJ_date.Hotlifetime THEN
    Mach_Control.WJ_b.Error[12]:=TRUE;//热切丝使用寿命到达
END_IF
END_ACTION

ACTION TailCurl_Auto_CamOut:
//判断是否有叠台部分轴在耦合中
				IF NOT arrAxisCtrl[AxiseNo.AxisName.TailCurlSEPTALine].Status.Coupled AND NOT arrAxisCtrl[AxiseNo.AxisName.TailCurlSEPTAUpDown].Status.Coupled AND 
					NOT arrAxisCtrl[AxiseNo.AxisName.SCurlingneedleWhirling].Status.Coupled AND NOT arrAxisCtrl[AxiseNo.AxisName.LCurlingneedleWhirling].Status.Coupled   THEN
					TailCurl_AxiseCoupling:=FALSE;//叠片部分轴在耦合中
				ELSE
					TailCurl_AxiseCoupling:=TRUE;
				END_IF
//叠台自动子程序_凸轮耦合解除_主轴清零
rWJCamOut_TRIG(CLK:=Mach_Control.WJ_b.WJ_AllCamOut , Q=> );
IF  rWJCamOut_TRIG.Q THEN
	TailCurl_Step1:=100;
END_IF
CASE TailCurl_Step1 OF
		100://先判断主轴是否在停止中
				IF arrAxisCtrl[AxiseNo.VirAxisName.VirTailCurl].Status.NoMoving  THEN
					arrAxisCtrl[AxiseNo.VirAxisName.VirTailCurl].Cmd.bStop:=FALSE;
					TailCurl_Step1:=110;
				ELSE
					arrAxisCtrl[AxiseNo.VirAxisName.VirTailCurl].Cmd.bStop:=TRUE;
				END_IF
		110://判断轴是否在耦合中
				//IF TailCurl_AxiseCoupling THEN
					TailCurl_Step1:=120;
				//ELSE
					//TailCurl_Step1:=130;
				//END_IF
		120://叠台部轴解除耦合
				fbCamInEndWindX.bCamInExecute:=FALSE;//夹膜平移
				fbCamInEndWindY.bCamInExecute:=FALSE;//夹膜升降
				tailCurl1_GearIn.Execute:=FALSE;//短卷针
				tailCurl2_GearIn.Execute:=FALSE;//长卷针
				tailCurlGearInEnable:=FALSE;//夹隔膜电子凸轮
				tailCurlGearInEnable1:=FALSE;//夹隔膜电子凸轮
				tailRetGearInEnable:=FALSE;//夹电芯平移与夹电芯伸缩电子齿轮
				IF NOT fbCamInEndWindX.bCamInExecute AND NOT fbCamInEndWindY.bCamInExecute AND 
					NOT  tailCurl1_GearIn.Execute AND NOT tailCurl2_GearIn.Execute AND NOT tailCurlGearInEnable AND NOT tailRetGearInEnable AND NOT tailCurlGearInEnable1  THEN
						TailCurl_Step1:=130;
				END_IF
		130:
				arrAxisCtrl[AxiseNo.AxisName.TailCurlSEPTALine].Cmd.bGearOut:=TRUE;
				arrAxisCtrl[AxiseNo.AxisName.TailCurlSEPTAUpDown].Cmd.bGearOut:=TRUE;
				arrAxisCtrl[AxiseNo.AxisName.SCurlingneedleWhirling].Cmd.bGearOut:=TRUE;
				arrAxisCtrl[AxiseNo.AxisName.LCurlingneedleWhirling].Cmd.bGearOut:=TRUE;
			
				IF NOT DT_AxiseCoupling THEN
					arrAxisCtrl[AxiseNo.AxisName.TailCurlSEPTALine].Cmd.bGearOut:=FALSE;
					arrAxisCtrl[AxiseNo.AxisName.TailCurlSEPTAUpDown].Cmd.bGearOut:=FALSE;
					arrAxisCtrl[AxiseNo.AxisName.SCurlingneedleWhirling].Cmd.bGearOut:=FALSE;
					arrAxisCtrl[AxiseNo.AxisName.LCurlingneedleWhirling].Cmd.bGearOut:=FALSE;
									
					TailCurl_Step1:=140;
				END_IF
		140://主轴当前位置清零				
				arrAxisCtrl[AxiseNo.VirAxisName.VirTailCurl].Cmd.fSetPos:=0;
				arrAxisCtrl[AxiseNo.VirAxisName.VirTailCurl].Cmd.bSetPos:=TRUE;			
				TailCurl_Step1:=150;
		150://判断主轴是否停止以及在模长初始位
				IF  NOT arrAxisCtrl[AxiseNo.VirAxisName.VirTailCurl].Cmd.bSetPos AND arrAxis[AxiseNo.VirAxisName.VirTailCurl].NcToPlc.SetPos=0   THEN
					TailCurl_Step1:=6666;
				END_IF
END_CASE
END_ACTION

ACTION TailCurl_Auto1:
//TON_TailCurl[0](PT:=T#0.5S);//热切加热延时时间
hot_time_ton(PT:=T#0.3S);
WJ_TON[1].PT:=REAL_TO_TIME(Par.stWJ_date.HotTime*1000);
SLCurlingneedleLine_TON(PT:=T#0.5S);
WJ_TON[6](IN:= , PT:=T#100MS , Q=> , ET=> );//
TON_TailCurl[1](IN:=Mach_Control.WJ_b.HotCut,PT:=T#0.4S);//热切丝加热时间
IF TON_TailCurl[1].Q THEN
	Mach_Control.WJ_b.HotCut:=FALSE;
	Par.stWJ_date.Hotcount:=Par.stWJ_date.Hotcount+1;
END_IF


IF WJ_TON[1].Q THEN//热切丝自动
	Mach_Control.WJ_b.HotCut:=FALSE;
	WJ_TON[1].IN:=FALSE;
END_IF

IF  Mach_Control.WJ_b.HotClear THEN
	Par.stWJ_date.Hotcount:=0;
END_IF

IF Mach_Control.U.WJ_iMode=3 THEN
	Mach_Control.WJ_b.Manual:=TRUE;
	ELSE
	Mach_Control.WJ_b.Manual:=FALSE;	
END_IF

/////////////////尾卷辅助时间计时////////////////////////
IF DP_Step0=6040  (*AND  NOT Mach_Control.DT_b.OffloadDone*) THEN
     Mach_Control.WJ_b.WJ_TIME:=(TIME_TO_REAL(WJ_ET))/1000;
END_IF	 
WJ_TON[2](IN:= (DP_Step0=6040 AND   Mach_Control.U.DT_iMode=1 AND  TailCurlStep3<=220 AND Mach_Control.U.WJ_iMode=1 ), PT:=T#500S, Q=> , ET=>WJ_ET );
/////////////////////////////////////////////////////////////

////////////////   
(*IF Blueflaging THEN
	Par.stDT_date.BH_Thickness :=0.5*(((Par.stDT_date.An_Thickness+Par.stDT_date.SEPTA_Thickness)*Par.stDT_date.An_Quantity+(Par.stDT_date.Ca_Thickness+Par.stDT_date.SEPTA_Thickness)*Par.stDT_date.Ca_Quantity)-((Par.stDT_date.An_Thickness+Par.stDT_date.SEPTA_Thickness)*(Mach_Control.An_b.An_Quantited-Mach_Control.An_b.An_EmptyRunKDQuantited)+(Par.stDT_date.Ca_Thickness+Par.stDT_date.SEPTA_Thickness)*(Mach_Control.Ca_b.Ca_Quantited-Mach_Control.Ca_b.Ca_EmptyRunKDQuantited))+(Mach_Control.An_b.An_EmptyRunKDQuantited +Mach_Control.Ca_b.Ca_EmptyRunKDQuantited )*Par.stDT_date.SEPTA_Thickness);
ELSE
	Par.stDT_date.BH_Thickness :=0.5*(((Par.stDT_date.An_Thickness+Par.stDT_date.SEPTA_Thickness)*Par.stDT_date.An_Quantity+(Par.stDT_date.Ca_Thickness+Par.stDT_date.SEPTA_Thickness)*Par.stDT_date.Ca_Quantity)-((Par.stDT_date.An_Thickness+Par.stDT_date.SEPTA_Thickness)*Mach_Control.An_b.An_Quantited+(Par.stDT_date.Ca_Thickness+Par.stDT_date.SEPTA_Thickness)*Mach_Control.Ca_b.Ca_Quantited));
END_IF
arrAxispar[AxiseNo.AxisName.TailCurlUpDown].arrTargetPoint[6]:=arrAxispar[AxiseNo.AxisName.TailCurlUpDown].arrTargetPoint[1]-Par.stDT_date.BH_Thickness;
arrAxispar[AxiseNo.AxisName.TailCurlSEPTAUpDown].arrTargetPoint[3]:=arrAxispar[AxiseNo.AxisName.TailCurlSEPTAUpDown].arrTargetPoint[1]+Par.stDT_date.BH_Thickness;	*)				
////////////////
IF Blueflaging AND NOT Mach_Control.U.EmptyRunMode THEN
	Par.stDT_date.BH_Thickness :=0.5*(((Par.stDT_date.An_Thickness+Par.stDT_date.SEPTA_Thickness)*Par.stDT_date.An_Quantity+(Par.stDT_date.Ca_Thickness+Par.stDT_date.SEPTA_Thickness)*Par.stDT_date.Ca_Quantity)-((Par.stDT_date.An_Thickness+Par.stDT_date.SEPTA_Thickness)*Mach_Control.An_b.An_Quantited+(Par.stDT_date.Ca_Thickness+Par.stDT_date.SEPTA_Thickness)*Mach_Control.Ca_b.Ca_Quantited)+40*Par.stDT_date.SEPTA_Thickness);
ELSIF NOT  Blueflaging AND NOT Mach_Control.U.EmptyRunMode THEN
	Par.stDT_date.BH_Thickness :=0.5*(((Par.stDT_date.An_Thickness+Par.stDT_date.SEPTA_Thickness)*Par.stDT_date.An_Quantity+(Par.stDT_date.Ca_Thickness+Par.stDT_date.SEPTA_Thickness)*Par.stDT_date.Ca_Quantity)-((Par.stDT_date.An_Thickness+Par.stDT_date.SEPTA_Thickness)*Mach_Control.An_b.An_Quantited+(Par.stDT_date.Ca_Thickness+Par.stDT_date.SEPTA_Thickness)*Mach_Control.Ca_b.Ca_Quantited));
ELSIF Mach_Control.U.EmptyRunMode THEN
	Par.stDT_date.BH_Thickness :=0.5*(((Par.stDT_date.An_Thickness+Par.stDT_date.SEPTA_Thickness)*Par.stDT_date.An_Quantity+(Par.stDT_date.Ca_Thickness+Par.stDT_date.SEPTA_Thickness)*Par.stDT_date.Ca_Quantity))-(Par.stDT_date.SEPTA_Thickness*(Mach_Control.An_b.An_Quantited+Mach_Control.Ca_b.Ca_Quantited));
END_IF
arrAxispar[AxiseNo.AxisName.TailCurlUpDown].arrTargetPoint[6]:=arrAxispar[AxiseNo.AxisName.TailCurlUpDown].arrTargetPoint[1]-Par.stDT_date.BH_Thickness;
arrAxispar[AxiseNo.AxisName.TailCurlSEPTAUpDown].arrTargetPoint[3]:=arrAxispar[AxiseNo.AxisName.TailCurlSEPTAUpDown].arrTargetPoint[1]+Par.stDT_date.BH_Thickness;	


IF (TailCurlStep3>=150 AND TailCurlStep3<=210) OR (TailCurlStep3>=1050 AND TailCurlStep3<=1140) THEN
	iTargetTorqueTest:=Par.stDT_date.iTargetTorqueHMI*Par.stDT_date.iTargetTorqueBLXS/10;
ELSIF  	(* Mach_Control.An_b.An_Quantited<1*) NOT  bFirstFoldFinish[1] OR (Mach_Control.Ca_b.Ca_Quantited= Par.stDT_date.Ca_Quantity  AND Mach_Control.An_b.An_Quantited= Par.stDT_date.An_Quantity) THEN
	iTargetTorqueTest:=Par.stDT_date.iTargetTorqueHMI*6/10;
ELSE
	iTargetTorqueTest:=Par.stDT_date.iTargetTorqueHMI;
END_IF


TON_TailCurl[2](PT:=T#0.5S);//长卷针夹爪气缸延时
TON_TailCurl[3](PT:=T#1S);//长卷针泄压时间
TON_TailCurl[4](PT:=T#0.5S);//短卷针夹爪气缸延时
TON_TailCurl[5](PT:=T#1S);//短卷针泄压时间
TON_TailCurl[6](PT:=T#1S);//短卷针泄压时间
TON_TailCurl1[2](PT:=T#0.2S);
TON_TailCurl1[3](PT:=T#1S);
TON_TailCurl1[4](PT:=T#0.2S);
TON_TailCurl1[5](PT:=T#0.2S);
TON_TailCurl1[6](PT:=T#0.3S);
TailCurlSplintCy_TON(PT:=T#2S);//夹NG料延时
TailCurlSplintCy_ON(PT:=T#1.5S);//夹NG料延时
//判断始尾卷各轴是否在初始位置
IF arrAxisCtrl[AxiseNo.AxisName.TailCurlLine].Cmd.arrbRealPoint[11] AND arrAxisCtrl[AxiseNo.AxisName.TailCurlRetracting].Cmd.arrbRealPoint[1] AND
	arrAxisCtrl[AxiseNo.AxisName.TailCurlUpDown].Cmd.arrbRealPoint[1] AND arrAxisCtrl[AxiseNo.AxisName.TailCurlSEPTALine].Cmd.arrbRealPoint[1] AND 
	 arrAxisCtrl[AxiseNo.AxisName.TailCurlSEPTAUpDown].Cmd.arrbRealPoint[1] AND arrAxisCtrl[AxiseNo.AxisName.LCurlingneedleWhirling].Cmd.arrbRealPoint[1] AND 
	arrAxisCtrl[AxiseNo.AxisName.SCurlingneedleWhirling].Cmd.arrbRealPoint[1] AND arrAxisCtrl[AxiseNo.AxisName.LCurlingneedleLine].Cmd.arrbRealPoint[1] AND 
	arrAxisCtrl[AxiseNo.AxisName.SCurlingneedleLine].Cmd.arrbRealPoint[1]  AND arrAxisCtrl[AxiseNo.AxisName.TailCurlWhirling].Cmd.arrbRealPoint[1] THEN
	TailCurlIinitPos:=TRUE;//尾卷各轴都在初始位
ELSE
	TailCurlIinitPos:=FALSE;	
END_IF
rWJ_SinStepd(CLK:=Mach_Control.WJ_b.TailCurlStart , Q=> );
IF rWJ_SinStepd.Q THEN
	TailCurlSinStep:=FALSE;
END_IF
(*
IF TailCurlStep3>=150 AND TailCurlStep3 <151 THEN
	arrAxisPar[AxiseNo.AxisName.TailCurlSEPTALine].fVelocity_of_Abs:=arrAxisPar[AxiseNo.AxisName.TailCurlLine].fVelocity_of_Abs*0.85;
ELSE
	arrAxisPar[AxiseNo.AxisName.TailCurlSEPTALine].fVelocity_of_Abs:=arrAxisPar[AxiseNo.AxisName.TailCurlLine].fVelocity_of_Abs;
END_IF
*)

//尾卷夹电芯拉膜速度切换
(*
IF TailCurlStep3>260 AND TailCurlStep3<1000 THEN
	arrAxisPar[AxiseNo.AxisName.TailCurlSEPTALine].fVelocity_of_Abs:=arrAxisPar[AxiseNo.AxisName.TailCurlSEPTALine].fVelocity_of_Abs;
	arrAxisPar[AxiseNo.AxisName.TailCurlLine].fVelocity_of_Abs:=arrAxisPar[AxiseNo.AxisName.TailCurlLine].fVelocity_of_Abs ;	
ELSIF(TailCurlStep3<=105  AND TailCurlStep3>=100)
	OR  (TailCurlStep3<=1010   AND TailCurlStep3>=1000)
	OR  (TailCurlStep3<=215 AND TailCurlStep3>=213) THEN
	arrAxisPar[AxiseNo.AxisName.TailCurlSEPTALine].fVelocity_of_Abs:=Par.stDT_date.fVelocity_of_QDX ;
	arrAxisPar[AxiseNo.AxisName.TailCurlLine].fVelocity_of_Abs:=Par.stDT_date.fVelocity_of_QDX ;
ELSE	
	arrAxisPar[AxiseNo.AxisName.TailCurlSEPTALine].fVelocity_of_Abs:=Par.stDT_date.fVelocity_of_LM ;
	arrAxisPar[AxiseNo.AxisName.TailCurlLine].fVelocity_of_Abs:=Par.stDT_date.fVelocity_of_LM ;
END_IF
*)
IF (TailCurlStep3<=190  AND TailCurlStep3>=145) OR (TailCurlStep3<=1060  AND TailCurlStep3>=1140) OR  (TailCurlStep3<215 AND TailCurlStep3>=213) THEN
	arrAxisPar[AxiseNo.AxisName.TailCurlSEPTALine].fVelocity_of_Abs:=Par.stDT_date.fVelocity_of_LM ;
	arrAxisPar[AxiseNo.AxisName.TailCurlLine].fVelocity_of_Abs:=Par.stDT_date.fVelocity_of_LM ;
ELSIF (TailCurlStep3<=105  AND TailCurlStep3>=100)OR  (TailCurlStep3<=1010   AND TailCurlStep3>=1000)  THEN
	arrAxisPar[AxiseNo.AxisName.TailCurlSEPTALine].fVelocity_of_Abs:=Par.stDT_date.fVelocity_of_QDX ;
	arrAxisPar[AxiseNo.AxisName.TailCurlLine].fVelocity_of_Abs:=Par.stDT_date.fVelocity_of_QDX ;
ELSE
	arrAxisPar[AxiseNo.AxisName.TailCurlSEPTALine].fVelocity_of_Abs:=Par.stDT_date.fVelocity_of_QDX ;
	arrAxisPar[AxiseNo.AxisName.TailCurlLine].fVelocity_of_Abs:=Par.stDT_date.fVelocity_of_QDX ;
END_IF



IF Mach_Control.U.WJ_iMode=1 THEN//在自动状态下
//尾卷取叠台电芯自动
		CASE TailCurlStep3 OF 
				0://判断叠台是否叠电芯完成
					IF  TailCurlIinitPos THEN//尾卷夹电芯平移在初始位、尾卷夹电芯伸缩在初始位
						
						arrAxisCtrl[AxiseNo.AxisName.TailCurlSEPTALine].Cmd.fOverride:=100;
						arrAxisCtrl[AxiseNo.AxisName.TailCurlRetracting].Cmd.fOverride:=100;
						arrAxisCtrl[AxiseNo.AxisName.TailCurlLine].Cmd.fOverride:=100;
				
						IF NOT CellMemory[Mach_Control.DT_b.DT_Memory].Overhang_TF AND NOT Mach_Control.WJ_b.b_WJqr AND Mach_Control.DT_b.OffloadRequest AND arrAxisCtrl[AxiseNo.AxisName.LCurlingneedleLine].Cmd.arrbRealPoint[1] 
							 AND arrAxisCtrl[AxiseNo.AxisName.SCurlingneedleLine].Cmd.arrbRealPoint[1] AND arrAxisCtrl[AxiseNo.AxisName.LCurlingneedleLine].Cmd.arrbRealPoint[1]
								AND arrAxisCtrl[AxiseNo.AxisName.SCurlingneedleWhirling].Cmd.arrbRealPoint[1]  AND   arrAxisCtrl[AxiseNo.AxisName.LCurlingneedleWhirling].Cmd.arrbRealPoint[1]
								AND arrAxisCtrl[AxiseNo.AxisName.TailCurlLine].Cmd.arrbRealPoint[11] AND arrAxisCtrl[AxiseNo.AxisName.TailCurlRetracting].Cmd.arrbRealPoint[1] 
								AND arrAxisCtrl[AxiseNo.AxisName.TailCurlSEPTALine].Cmd.arrbRealPoint[1] AND arrAxisCtrl[AxiseNo.AxisName.TailCurlWhirling].Cmd.arrbRealPoint[1] THEN
								
								TailCurlStep3:=100;//正常尾卷流程
								IF Mach_Control.WJ_b.SinStepMode THEN//尾卷单步模式
									TailCurlSinStep:=TRUE;
								ELSE
									TailCurlSinStep:=FALSE;
								END_IF	
						ELSIF NOT CellMemory[Mach_Control.DT_b.DT_Memory].Overhang_TF  AND  Mach_Control.WJ_b.b_WJqr AND Mach_Control.DT_b.OffloadRequest AND arrAxisCtrl[AxiseNo.AxisName.LCurlingneedleLine].Cmd.arrbRealPoint[1] 
							AND arrAxisCtrl[AxiseNo.AxisName.SCurlingneedleLine].Cmd.arrbRealPoint[1] AND arrAxisCtrl[AxiseNo.AxisName.LCurlingneedleLine].Cmd.arrbRealPoint[1]
							AND arrAxisCtrl[AxiseNo.AxisName.SCurlingneedleWhirling].Cmd.arrbRealPoint[1]  AND   arrAxisCtrl[AxiseNo.AxisName.LCurlingneedleWhirling].Cmd.arrbRealPoint[1] 
							AND arrAxisCtrl[AxiseNo.AxisName.TailCurlLine].Cmd.arrbRealPoint[11] AND arrAxisCtrl[AxiseNo.AxisName.TailCurlRetracting].Cmd.arrbRealPoint[1] 
							AND arrAxisCtrl[AxiseNo.AxisName.TailCurlSEPTALine].Cmd.arrbRealPoint[1] AND arrAxisCtrl[AxiseNo.AxisName.TailCurlWhirling].Cmd.arrbRealPoint[1] THEN
							
								TailCurlStep3:=900;//NG尾卷流程
							IF Mach_Control.WJ_b.SinStepMode THEN//尾卷单步模式
								TailCurlSinStep:=TRUE;
							ELSE
								TailCurlSinStep:=FALSE;
							END_IF		
						ELSIF	CellMemory[Mach_Control.DT_b.DT_Memory].Overhang_TF AND Mach_Control.DT_b.OffloadRequest AND arrAxisCtrl[AxiseNo.AxisName.LCurlingneedleLine].Cmd.arrbRealPoint[1] 
							 AND arrAxisCtrl[AxiseNo.AxisName.SCurlingneedleLine].Cmd.arrbRealPoint[1] AND arrAxisCtrl[AxiseNo.AxisName.LCurlingneedleLine].Cmd.arrbRealPoint[1]
								AND arrAxisCtrl[AxiseNo.AxisName.SCurlingneedleWhirling].Cmd.arrbRealPoint[1]  AND   arrAxisCtrl[AxiseNo.AxisName.LCurlingneedleWhirling].Cmd.arrbRealPoint[1] 
								AND arrAxisCtrl[AxiseNo.AxisName.TailCurlLine].Cmd.arrbRealPoint[11] AND arrAxisCtrl[AxiseNo.AxisName.TailCurlRetracting].Cmd.arrbRealPoint[1] 
								AND arrAxisCtrl[AxiseNo.AxisName.TailCurlSEPTALine].Cmd.arrbRealPoint[1] AND arrAxisCtrl[AxiseNo.AxisName.TailCurlWhirling].Cmd.arrbRealPoint[1] THEN	
									
									TailCurlStep3:=1000;//对齐度NG不尾卷流程
								IF Mach_Control.WJ_b.SinStepMode THEN//尾卷单步模式
									TailCurlSinStep:=TRUE;
								ELSE
									TailCurlSinStep:=FALSE;
								END_IF								
							END_IF	
						ELSE
							IF Mach_Control.WJ_b.SinStepMode THEN//尾卷单步模式
								TailCurlSinStep:=TRUE;
							ELSE
								TailCurlSinStep:=FALSE;
							END_IF						
							TailCurlStep3:=10;	
						END_IF
	
				10://尾卷夹电芯气缸张开
							IF NOT TailCurlSinStep  THEN
									//arrCyCtrl[arrCyNo.CylinderName.CurlingSplintCy_S_1].Cmd.bON:=TRUE;//尾卷短卷针泄压关闭
									arrCyCtrl[arrCyNo.CylinderName.TailCurlSplintCy].Cmd.bOFF:=TRUE;//尾卷取料夹爪气缸张开	
									arrCyCtrl[arrCyNo.CylinderName.CurlingSplintCy_L].Cmd.bOFF:=TRUE;//尾卷长卷针张开
									arrCyCtrl[arrCyNo.CylinderName.CurlingSplintCy_S].Cmd.bOFF:=TRUE;//尾卷短卷针张开	
									arrCyCtrl[arrCyNo.CylinderName.PoleHotCutterCy].Cmd.bOFF:=TRUE;//隔膜热切升降气缸收回
									arrCyCtrl[arrCyNo.CylinderName.PoleSplintCy_D].Cmd.bOFF:=TRUE;//隔膜隔膜下夹板气缸收回						
									arrCyCtrl[arrCyNo.CylinderName.TailCurlUpdownCy].Cmd.bOFF:=TRUE;//尾卷压轮升降气缸收回
									IF arrCyCtrl[arrCyNo.CylinderName.TailCurlUpdownCy].Io.DIOFFSwitch THEN
										arrCyCtrl[arrCyNo.CylinderName.TailCurlLineCy].Cmd.bOFF:=TRUE;//尾卷压轮平移气缸收回	
									END_IF						
									IF arrCyCtrl[arrCyNo.CylinderName.TailCurlSplintCy].Status.OFFState AND arrCyCtrl[arrCyNo.CylinderName.PoleHotCutterCy].Status.OFFState AND arrCyCtrl[arrCyNo.CylinderName.PoleSplintCy_D].Status.OFFState AND
										 arrCyCtrl[arrCyNo.CylinderName.TailCurlUpdownCy].Status.OFFState AND arrCyCtrl[arrCyNo.CylinderName.TailCurlLineCy].Status.OFFState THEN
										IF Mach_Control.WJ_b.SinStepMode THEN//尾卷单步模式
											TailCurlSinStep:=TRUE;
										ELSE
											TailCurlSinStep:=FALSE;
										END_IF
										TailCurlStep3:=20;	
									END_IF
							END_IF
				20://
					IF NOT TailCurlSinStep THEN
							//长卷针平移至初始位
							IF 	arrAxisCtrl[AxiseNo.AxisName.LCurlingneedleLine].Status.Homed AND arrAxisCtrl[AxiseNo.AxisName.LCurlingneedleLine].Status.NoMoving THEN
								IF arrAxisCtrl[AxiseNo.AxisName.LCurlingneedleLine].Cmd.arrbRealPoint[1] THEN
									arrAxisCtrl[AxiseNo.AxisName.LCurlingneedleLine].Cmd.iGoSetPos:=0;
								ELSE
									arrAxisCtrl[AxiseNo.AxisName.LCurlingneedleLine].Cmd.iGoSetPos:=1;
								END_IF
							END_IF
							//短卷针平移至初始位
							IF 	arrAxisCtrl[AxiseNo.AxisName.SCurlingneedleLine].Status.Homed AND arrAxisCtrl[AxiseNo.AxisName.SCurlingneedleLine].Status.NoMoving THEN
								IF arrAxisCtrl[AxiseNo.AxisName.SCurlingneedleLine].Cmd.arrbRealPoint[1] THEN
									arrAxisCtrl[AxiseNo.AxisName.SCurlingneedleLine].Cmd.iGoSetPos:=0;
								ELSE
									arrAxisCtrl[AxiseNo.AxisName.SCurlingneedleLine].Cmd.iGoSetPos:=1;
								END_IF
							END_IF		
							IF 	arrAxisCtrl[AxiseNo.AxisName.LCurlingneedleLine].Cmd.arrbRealPoint[1]  AND arrAxisCtrl[AxiseNo.AxisName.SCurlingneedleLine].Cmd.arrbRealPoint[1] THEN
								IF Mach_Control.WJ_b.SinStepMode THEN//尾卷单步模式
									TailCurlSinStep:=TRUE;
								ELSE
									TailCurlSinStep:=FALSE;
								END_IF								
								TailCurlStep3:=30;	
							END_IF
					END_IF
				30://尾卷夹电芯平移、夹电芯伸缩移动至初始位
					IF NOT TailCurlSinStep THEN
							//尾卷夹电芯平移
							IF 	arrAxisCtrl[AxiseNo.AxisName.TailCurlLine].Status.Homed AND arrAxisCtrl[AxiseNo.AxisName.TailCurlLine].Status.NoMoving AND 
                                    arrAxisCtrl[AxiseNo.AxisName.LCurlingneedleLine].Cmd.arrbRealPoint[1]  AND arrAxisCtrl[AxiseNo.AxisName.SCurlingneedleLine].Cmd.arrbRealPoint[1]      THEN
								IF arrAxisCtrl[AxiseNo.AxisName.TailCurlLine].Cmd.arrbRealPoint[1] THEN
									arrAxisCtrl[AxiseNo.AxisName.TailCurlLine].Cmd.iGoSetPos:=0;
								ELSE
									arrAxisCtrl[AxiseNo.AxisName.TailCurlLine].Cmd.iGoSetPos:=1;
								END_IF
							END_IF
							//尾卷夹电芯伸缩
							IF 	arrAxisCtrl[AxiseNo.AxisName.TailCurlRetracting].Status.Homed AND arrAxisCtrl[AxiseNo.AxisName.TailCurlRetracting].Status.NoMoving THEN
								IF arrAxisCtrl[AxiseNo.AxisName.TailCurlRetracting].Cmd.arrbRealPoint[1] THEN
									//TailCurlRetMark:=FALSE;//尾卷夹电芯伸缩力矩判断标志
									arrAxisCtrl[AxiseNo.AxisName.TailCurlRetracting].Cmd.iGoSetPos:=0;
								ELSE
									arrAxisCtrl[AxiseNo.AxisName.TailCurlRetracting].Cmd.iGoSetPos:=1;
									//TailCurlRetMark:=TRUE;//尾卷夹电芯伸缩力矩判断标志
								END_IF
							END_IF	
							//尾卷夹电芯升降
							IF 	arrAxisCtrl[AxiseNo.AxisName.TailCurlUpDown].Status.Homed AND arrAxisCtrl[AxiseNo.AxisName.TailCurlUpDown].Status.NoMoving THEN
								IF arrAxisCtrl[AxiseNo.AxisName.TailCurlUpDown].Cmd.arrbRealPoint[1] THEN
									arrAxisCtrl[AxiseNo.AxisName.TailCurlUpDown].Cmd.iGoSetPos:=0;
								ELSE
									arrAxisCtrl[AxiseNo.AxisName.TailCurlUpDown].Cmd.iGoSetPos:=1;
								END_IF
							END_IF
							//尾卷夹隔膜平移
							IF 	arrAxis[AxiseNo.AxisName.TailCurlSEPTALine].Status.Homed AND arrAxisCtrl[AxiseNo.AxisName.TailCurlSEPTALine].Status.NoMoving THEN
								IF arrAxisCtrl[AxiseNo.AxisName.TailCurlSEPTALine].Cmd.arrbRealPoint[1] THEN
									arrAxisCtrl[AxiseNo.AxisName.TailCurlSEPTALine].Cmd.iGoSetPos:=0;
								ELSE
									arrAxisCtrl[AxiseNo.AxisName.TailCurlSEPTALine].Cmd.iGoSetPos:=1;
								END_IF
							END_IF	
							//	尾卷夹隔膜升降
								IF 	arrAxisCtrl[AxiseNo.AxisName.TailCurlSEPTAUpDown].Status.Homed AND arrAxisCtrl[AxiseNo.AxisName.TailCurlSEPTAUpDown].Status.NoMoving THEN
								IF arrAxisCtrl[AxiseNo.AxisName.TailCurlSEPTAUpDown].Cmd.arrbRealPoint[1] THEN
									arrAxisCtrl[AxiseNo.AxisName.TailCurlSEPTAUpDown].Cmd.iGoSetPos:=0;
								ELSE
									arrAxisCtrl[AxiseNo.AxisName.TailCurlSEPTAUpDown].Cmd.iGoSetPos:=1;
								END_IF
							END_IF							
							//尾卷长卷针旋转
							IF 	arrAxisCtrl[AxiseNo.AxisName.LCurlingneedleWhirling].Status.Homed AND arrAxisCtrl[AxiseNo.AxisName.LCurlingneedleWhirling].Status.NoMoving THEN
								IF arrAxisCtrl[AxiseNo.AxisName.LCurlingneedleWhirling].Cmd.arrbRealPoint[1] THEN
									arrAxisCtrl[AxiseNo.AxisName.LCurlingneedleWhirling].Cmd.iGoSetPos:=0;
								ELSE
									arrAxisCtrl[AxiseNo.AxisName.LCurlingneedleWhirling].Cmd.iGoSetPos:=1;
								END_IF
							END_IF	
							//尾卷短卷针旋转
							IF 	arrAxisCtrl[AxiseNo.AxisName.SCurlingneedleWhirling].Status.Homed AND arrAxisCtrl[AxiseNo.AxisName.SCurlingneedleWhirling].Status.NoMoving THEN
								IF arrAxisCtrl[AxiseNo.AxisName.SCurlingneedleWhirling].Cmd.arrbRealPoint[1] THEN
									arrAxisCtrl[AxiseNo.AxisName.SCurlingneedleWhirling].Cmd.iGoSetPos:=0;
								ELSE
									arrAxisCtrl[AxiseNo.AxisName.SCurlingneedleWhirling].Cmd.iGoSetPos:=1;
								END_IF
							END_IF							
							IF arrAxisCtrl[AxiseNo.AxisName.TailCurlLine].Cmd.arrbRealPoint[1] AND arrAxisCtrl[AxiseNo.AxisName.TailCurlRetracting].Cmd.arrbRealPoint[1] AND
								arrAxisCtrl[AxiseNo.AxisName.TailCurlUpDown].Cmd.arrbRealPoint[1] AND arrAxisCtrl[AxiseNo.AxisName.TailCurlSEPTALine].Cmd.arrbRealPoint[1] AND 
								 arrAxisCtrl[AxiseNo.AxisName.TailCurlSEPTAUpDown].Cmd.arrbRealPoint[1] AND arrAxisCtrl[AxiseNo.AxisName.LCurlingneedleWhirling].Cmd.arrbRealPoint[1] AND arrAxisCtrl[AxiseNo.AxisName.SCurlingneedleWhirling].Cmd.arrbRealPoint[1] THEN
								IF Mach_Control.WJ_b.SinStepMode THEN//尾卷单步模式
									TailCurlSinStep:=TRUE;
								ELSE
									TailCurlSinStep:=FALSE;
								END_IF							
								TailCurlStep3:=40;	
							END_IF
					END_IF
				40://尾卷夹旋转到取叠台电芯角度
					IF NOT TailCurlSinStep THEN
							IF 	arrAxis[AxiseNo.AxisName.TailCurlWhirling].Status.Homed AND arrAxisCtrl[AxiseNo.AxisName.TailCurlWhirling].Status.NoMoving AND 
								 arrAxisCtrl[AxiseNo.AxisName.TailCurlLine].Status.Homed AND arrAxisCtrl[AxiseNo.AxisName.TailCurlLine].Status.NoMoving AND arrAxisCtrl[AxiseNo.AxisName.TailCurlLine].Cmd.arrbRealPoint[1] AND 
								 arrAxisCtrl[AxiseNo.AxisName.TailCurlRetracting].Status.Homed AND arrAxisCtrl[AxiseNo.AxisName.TailCurlRetracting].Status.NoMoving AND arrAxisCtrl[AxiseNo.AxisName.TailCurlRetracting].Cmd.arrbRealPoint[1] THEN
										IF arrAxisCtrl[AxiseNo.AxisName.TailCurlWhirling].Cmd.arrbRealPoint[1] THEN
											arrAxisCtrl[AxiseNo.AxisName.TailCurlWhirling].Cmd.iGoSetPos:=0;
											IF Mach_Control.WJ_b.SinStepMode THEN//尾卷单步模式
												TailCurlSinStep:=TRUE;
											ELSE
												TailCurlSinStep:=FALSE;
											END_IF	
											TailCurlStep3:=50;	
										ELSE
											arrAxisCtrl[AxiseNo.AxisName.TailCurlWhirling].Cmd.iGoSetPos:=1;
										END_IF
							END_IF		
					END_IF
	            50://尾卷夹电芯平移去取电芯等待位
				     IF NOT TailCurlSinStep THEN
						   IF arrAxisCtrl[AxiseNo.AxisName.TailCurlWhirling].Cmd.arrbRealPoint[1] AND arrAxisCtrl[AxiseNo.AxisName.TailCurlUpDown].Cmd.arrbRealPoint[1] AND
							  arrAxisCtrl[AxiseNo.AxisName.TailCurlSEPTALine].Cmd.arrbRealPoint[1] AND  arrAxisCtrl[AxiseNo.AxisName.TailCurlSEPTAUpDown].Cmd.arrbRealPoint[1] AND
							  arrAxisCtrl[AxiseNo.AxisName.LCurlingneedleLine].Cmd.arrbRealPoint[1] AND arrAxisCtrl[AxiseNo.AxisName.SCurlingneedleLine].Cmd.arrbRealPoint[1] AND
							  arrCyCtrl[arrCyNo.CylinderName.PoleSplintCy_D].Io.DIOFFSwitch AND arrCyCtrl[arrCyNo.CylinderName.TailCurlUpdownCy].Io.DIOFFSwitch AND
							  arrAxisCtrl[AxiseNo.AxisName.TailCurlLine].Status.Homed AND arrAxisCtrl[AxiseNo.AxisName.TailCurlLine].Status.NoMoving  THEN
								   IF arrAxisCtrl[AxiseNo.AxisName.TailCurlLine].Cmd.arrbRealPoint[11]  THEN
									  arrAxisCtrl[AxiseNo.AxisName.TailCurlLine].Cmd.iGoSetPos:=0;
										IF Mach_Control.WJ_b.SinStepMode THEN//尾卷单步模式
										   TailCurlSinStep:=TRUE;
										ELSE
										   TailCurlSinStep:=FALSE;
										END_IF									
										   TailCurlStep3:=0;
										   TailCurlTorMark:=FALSE;//尾卷夹电芯平移力矩判断标志位
								   ELSE
									   arrAxisCtrl[AxiseNo.AxisName.TailCurlLine].Cmd.iGoSetPos:=11;//尾卷夹电芯平移去取电芯等待位
									   TailCurlTorMark:=TRUE;//尾卷夹电芯平移力矩判断标志位
								   END_IF   
							END_IF
	                  END_IF
	
	
			100://夹膜升降去取电芯位，夹电芯升降去取电芯位	///////////////////////////////////////////////
						//Mach_Control.DT_b.OffloadRequest:=FALSE;//复位电芯下料请求
					    IF NOT TailCurlSinStep THEN
							
							IF Mach_Control.DT_b.OffloadRequest AND DP_Step0=6040 THEN
									IF 	arrAxisCtrl[AxiseNo.AxisName.TailCurlUpDown].Status.Homed AND arrAxisCtrl[AxiseNo.AxisName.TailCurlUpDown].Status.NoMoving THEN
										IF arrAxisCtrl[AxiseNo.AxisName.TailCurlUpDown].Cmd.arrbRealPoint[1] THEN
											arrAxisCtrl[AxiseNo.AxisName.TailCurlUpDown].Cmd.iGoSetPos:=0;
										ELSE
											arrAxisCtrl[AxiseNo.AxisName.TailCurlUpDown].Cmd.iGoSetPos:=1;
										END_IF
									END_IF	
									IF 	arrAxisCtrl[AxiseNo.AxisName.TailCurlSEPTAUpDown].Status.Homed AND arrAxisCtrl[AxiseNo.AxisName.TailCurlSEPTAUpDown].Status.NoMoving THEN
										IF arrAxisCtrl[AxiseNo.AxisName.TailCurlSEPTAUpDown].Cmd.arrbRealPoint[1] THEN
											arrAxisCtrl[AxiseNo.AxisName.TailCurlSEPTAUpDown].Cmd.iGoSetPos:=0;
										ELSE
											arrAxisCtrl[AxiseNo.AxisName.TailCurlSEPTAUpDown].Cmd.iGoSetPos:=1;
										END_IF
									END_IF	
									IF 	arrAxisCtrl[AxiseNo.AxisName.TailCurlUpDown].Cmd.arrbRealPoint[1]  AND arrAxisCtrl[AxiseNo.AxisName.TailCurlUpDown].Cmd.arrbRealPoint[1] 
										AND arrAxisCtrl[AxiseNo.AxisName.TailCurlSEPTAUpDown].Cmd.arrbRealPoint[1]  AND arrAxisCtrl[AxiseNo.AxisName.TailCurlSEPTAUpDown].Cmd.arrbRealPoint[1]	THEN
										IF Mach_Control.WJ_b.SinStepMode THEN//尾卷单步模式
											TailCurlSinStep:=TRUE;
										ELSE
											TailCurlSinStep:=FALSE;
										END_IF								
										TailCurlStep3:=105;	
										TON_TailCurl[6].IN:=FALSE;
									END_IF
							ELSE
									TailCurlStep3:=0;
							END_IF		
						END_IF
					
		
					
				105://负极叠片搬运平移轴在安全位置，尾卷夹电芯平移至取电芯位 、尾卷夹电芯伸缩至取电芯位 、尾卷夹膜平移至隔膜切断位///////////////////
						IF NOT TailCurlSinStep AND arrAxisCtrl[AxiseNo.AxisName.CaDTCarryingLine].Cmd.arrbRealPoint[1] AND arrAxisCtrl[AxiseNo.AxisName.CaDTCarryingUpDown].Cmd.arrbRealPoint[5] AND
                             arrAxisCtrl[AxiseNo.AxisName.TailCurlWhirling].Cmd.arrbRealPoint[1] AND arrAxisCtrl[AxiseNo.AxisName.SEPTATLine].Cmd.arrbRealPoint[1] AND
							 arrAxisCtrl[AxiseNo.AxisName.TailCurlSEPTAUpDown].Cmd.arrbRealPoint[1] AND arrAxisCtrl[AxiseNo.AxisName.TailCurlUpDown].Cmd.arrbRealPoint[1] AND
							  arrAxisCtrl[AxiseNo.AxisName.LCurlingneedleLine].Cmd.arrbRealPoint[1]  AND arrAxisCtrl[AxiseNo.AxisName.SCurlingneedleLine].Cmd.arrbRealPoint[1]   AND
							arrCyCtrl[arrCyNo.CylinderName.TailCurlSplintCy].Status.OFFState AND arrCyCtrl[arrCyNo.CylinderName.PoleSplintCy_D].Status.OFFState  AND
                            arrCyCtrl[arrCyNo.CylinderName.PoleHotCutterCy].Status.OFFState THEN  
                 
								IF  Mach_Control.DT_b.OffloadRequest THEN	
									TailCurlStep3:=106;
									(*
											arrAxisCtrl[AxiseNo.AxisName.TailCurlSEPTALine].Cmd.fOverride:=100;
											arrAxisCtrl[AxiseNo.AxisName.TailCurlRetracting].Cmd.fOverride:=100;
											arrAxisCtrl[AxiseNo.AxisName.TailCurlLine].Cmd.fOverride:=95;
			
											IF   arrAxis[AxiseNo.AxisName.TailCurlSEPTALine].Status.Homed AND arrAxisCtrl[AxiseNo.AxisName.TailCurlSEPTALine].Status.NoMoving THEN
												IF arrAxisCtrl[AxiseNo.AxisName.TailCurlSEPTALine].Cmd.arrbRealPoint[2] THEN
													TailCurlSEPTATorMark:=FALSE;//夹膜平移力矩判断标志
													arrAxisCtrl[AxiseNo.AxisName.TailCurlSEPTALine].Cmd.iGoSetPos:=0;
												ELSE
													arrAxisCtrl[AxiseNo.AxisName.TailCurlSEPTALine].Cmd.iGoSetPos:=2;//尾卷夹隔膜平移取芯位
													TailCurlSEPTATorMark:=TRUE;//夹膜平移力矩判断标志
												END_IF
											END_IF
											IF 	arrAxisCtrl[AxiseNo.AxisName.TailCurlRetracting].Status.Homed AND arrAxisCtrl[AxiseNo.AxisName.TailCurlRetracting].Status.NoMoving THEN
												IF arrAxisCtrl[AxiseNo.AxisName.TailCurlRetracting].Cmd.arrbRealPoint[2] THEN
													arrAxisCtrl[AxiseNo.AxisName.TailCurlRetracting].Cmd.iGoSetPos:=0;
												ELSE
													arrAxisCtrl[AxiseNo.AxisName.TailCurlRetracting].Cmd.iGoSetPos:=2;//尾卷夹电芯伸缩至取电芯位
													//TailCurlRetMark:=TRUE;//尾卷夹电芯伸缩力矩判断标志
												END_IF
											END_IF					
											IF 	arrAxisCtrl[AxiseNo.AxisName.TailCurlLine].Status.Homed AND arrAxisCtrl[AxiseNo.AxisName.TailCurlLine].Status.NoMoving THEN
												IF arrAxisCtrl[AxiseNo.AxisName.TailCurlLine].Cmd.arrbRealPoint[2] THEN
													TailCurlTorMark:=FALSE;//尾卷夹电芯平移力矩判断标志位
													arrAxisCtrl[AxiseNo.AxisName.TailCurlLine].Cmd.iGoSetPos:=0;
												ELSE
													arrAxisCtrl[AxiseNo.AxisName.TailCurlLine].Cmd.iGoSetPos:=2;//尾卷夹电芯平移至取电芯位
													TailCurlTorMark:=TRUE;//尾卷夹电芯平移力矩判断标志位
												END_IF
											END_IF						
											IF arrAxisCtrl[AxiseNo.AxisName.TailCurlSEPTALine].Cmd.arrbRealPoint[2] AND arrAxisCtrl[AxiseNo.AxisName.TailCurlRetracting].Cmd.arrbRealPoint[2] AND
												arrAxisCtrl[AxiseNo.AxisName.TailCurlLine].Cmd.arrbRealPoint[2]  THEN
												//TailCurlRetMark:=FALSE;//尾卷夹电芯伸缩力矩判断标志
												IF  Mach_Control.WJ_b.SinStepMode THEN//尾卷单步模式
													TailCurlSinStep:=TRUE;
												ELSE
													TailCurlSinStep:=FALSE;
												END_IF	
												TailCurlStep3:=110;
												TailCurlSplintCy_ON.IN:=FALSE;
											END_IF
										*)
								ELSE				
										TailCurlStep3:=0;
								END_IF	
						ELSE
										Mach_Control.WJ_b.Error[11]:=TRUE;	//尾卷夹电芯平移至取电芯位时条件不满足报警			
						END_IF	
				106:
					tailCurlGearInEnable1:=TRUE;//夹电芯平移与夹膜平移电子齿轮----取料
					tailRetGearInEnable:=TRUE;//夹电芯平移与夹电芯伸缩电子齿轮
					IF tailCurl_GearIn1.InGear AND tailRetGearIn.InGear THEN
						TailCurlStep3:=107;
					END_IF			
				107:
					IF 	arrAxisCtrl[AxiseNo.AxisName.TailCurlLine].Status.Homed AND 
                           arrAxisCtrl[AxiseNo.AxisName.CaDTCarryingLine].Cmd.arrbRealPoint[1] AND arrAxisCtrl[AxiseNo.AxisName.CaDTCarryingUpDown].Cmd.arrbRealPoint[5] AND
                             arrAxisCtrl[AxiseNo.AxisName.TailCurlWhirling].Cmd.arrbRealPoint[1] AND arrAxisCtrl[AxiseNo.AxisName.SEPTATLine].Cmd.arrbRealPoint[1] AND
							 arrAxisCtrl[AxiseNo.AxisName.TailCurlSEPTAUpDown].Cmd.arrbRealPoint[1] AND arrAxisCtrl[AxiseNo.AxisName.TailCurlUpDown].Cmd.arrbRealPoint[1] AND
							  arrAxisCtrl[AxiseNo.AxisName.LCurlingneedleLine].Cmd.arrbRealPoint[1]  AND arrAxisCtrl[AxiseNo.AxisName.SCurlingneedleLine].Cmd.arrbRealPoint[1]   AND
							arrCyCtrl[arrCyNo.CylinderName.TailCurlSplintCy].Status.OFFState AND arrCyCtrl[arrCyNo.CylinderName.PoleSplintCy_D].Status.OFFState  AND
                            arrCyCtrl[arrCyNo.CylinderName.PoleHotCutterCy].Status.OFFState   THEN
								IF arrAxisCtrl[AxiseNo.AxisName.TailCurlLine].Cmd.arrbRealPoint[2 ] AND arrAxisCtrl[AxiseNo.AxisName.TailCurlLine].Status.NoMoving   THEN
									TailCurlTorMark:=FALSE;//尾卷夹电芯平移力矩判断标志位
									arrAxisCtrl[AxiseNo.AxisName.TailCurlLine].Cmd.iGoSetPos:=0;
									TailCurlStep3:=108;
								ELSE
									arrAxisCtrl[AxiseNo.AxisName.TailCurlLine].Cmd.iGoSetPos:=2;//尾卷夹电芯平移至取电芯位
									TailCurlTorMark:=TRUE;//尾卷夹电芯平移力矩判断标志位
								END_IF
					ELSE
										Mach_Control.WJ_b.Error[11]:=TRUE;	//尾卷夹电芯平移至取电芯位时条件不满足报警								
					END_IF		
				108:
					IF arrAxisCtrl[AxiseNo.AxisName.TailCurlSEPTALine].Cmd.arrbRealPoint[2] AND arrAxisCtrl[AxiseNo.AxisName.TailCurlRetracting].Cmd.arrbRealPoint[2] AND
						arrAxisCtrl[AxiseNo.AxisName.TailCurlLine].Cmd.arrbRealPoint[2]   THEN
						tailCurlGearInEnable1:=FALSE;//夹电芯平移与夹膜平移电子齿轮----取料
						tailRetGearInEnable:=FALSE;//夹电芯平移与夹电芯伸缩电子齿轮
					END_IF
					IF NOT tailCurl_GearIn1.InGear AND NOT tailRetGearIn.InGear THEN
						TailCurlStep3:=110;
					END_IF			
	
				110://尾卷夹电芯气缸夹紧//////////////////////////////
				
						arrAxisCtrl[AxiseNo.AxisName.TailCurlSEPTALine].Cmd.fOverride:=100;
						arrAxisCtrl[AxiseNo.AxisName.TailCurlRetracting].Cmd.fOverride:=100;
						arrAxisCtrl[AxiseNo.AxisName.TailCurlLine].Cmd.fOverride:=100;
				     
						IF NOT TailCurlSinStep THEN					
							arrCyCtrl[arrCyNo.CylinderName.TailCurlSplintCy].Cmd.bON:=TRUE;//尾卷取料夹爪气缸夹紧
							TailCurlSplintCy_ON.IN:=TRUE;				
							IF (*arrCyCtrl[arrCyNo.CylinderName.TailCurlSplintCy].Io.DIOnSwitch OR*) TailCurlSplintCy_ON.Q THEN
								IF Mach_Control.WJ_b.SinStepMode THEN//尾卷单步模式
									TailCurlSinStep:=TRUE;
								ELSE
									TailCurlSinStep:=FALSE;
								END_IF								
								TailCurlStep3:=120;
								TailCurlSplintCy_ON.IN:=FALSE;
								 Mach_Control.DT_b.OffloadRequest:=FALSE;//复位电芯下料请求
							END_IF
						END_IF
				120://叠台升降下降至下电芯位	
					IF NOT TailCurlSinStep THEN				
								IF 	arrAxisCtrl[AxiseNo.AxisName.DTUpDown].Status.Homed   THEN
										arrAxisCtrl[AxiseNo.AxisName.DTUpDown].Cmd.bHome:=FALSE;//叠台升降下降至下电芯位回原点
												IF arrAxisCtrl[AxiseNo.AxisName.DTUpDown].Status.NoMoving THEN
															IF arrAxisCtrl[AxiseNo.AxisName.DTUpDown].Cmd.arrbRealPoint[2] THEN
																arrAxisCtrl[AxiseNo.AxisName.DTUpDown].Cmd.iGoSetPos:=0;
																IF Mach_Control.WJ_b.SinStepMode THEN//尾卷单步模式
																	TailCurlSinStep:=TRUE;
																ELSE
																	TailCurlSinStep:=FALSE;
																END_IF									
																TailCurlStep3:=130;
															ELSE
																arrAxisCtrl[AxiseNo.AxisName.DTUpDown].Cmd.iGoSetPos:=2;//叠台升降下降至下电芯位
															END_IF
											END_IF
								ELSE
										arrAxisCtrl[AxiseNo.AxisName.DTUpDown].Cmd.bHome:=TRUE;//叠台升降下降至下电芯位回原点
								END_IF	
					END_IF
				130://左、右压刀升降轴上升至抽刀高度
						IF NOT TailCurlSinStep THEN						
							IF 	arrAxisCtrl[AxiseNo.AxisName.LeftYDUpDown].Status.Homed AND arrAxisCtrl[AxiseNo.AxisName.LeftYDUpDown].Status.NoMoving THEN
									IF arrAxisCtrl[AxiseNo.AxisName.LeftYDUpDown].Cmd.arrbRealPoint[4] THEN
										arrAxisCtrl[AxiseNo.AxisName.LeftYDUpDown].Cmd.iGoSetPos:=0;
									ELSE
										arrAxisCtrl[AxiseNo.AxisName.LeftYDUpDown].Cmd.iGoSetPos:=4;//左压刀升降轴上升至抽刀高度
									END_IF
								END_IF					
								IF 	arrAxisCtrl[AxiseNo.AxisName.RightYDUpDown].Status.Homed AND arrAxisCtrl[AxiseNo.AxisName.RightYDUpDown].Status.NoMoving THEN
									IF arrAxisCtrl[AxiseNo.AxisName.RightYDUpDown].Cmd.arrbRealPoint[4] THEN
										arrAxisCtrl[AxiseNo.AxisName.RightYDUpDown].Cmd.iGoSetPos:=0;
									ELSE
										arrAxisCtrl[AxiseNo.AxisName.RightYDUpDown].Cmd.iGoSetPos:=4;//右压好升降上升至抽刀高度
									END_IF
								END_IF				
								IF arrAxisCtrl[AxiseNo.AxisName.LeftYDUpDown].Cmd.arrbRealPoint[4] AND arrAxisCtrl[AxiseNo.AxisName.RightYDUpDown].Cmd.arrbRealPoint[4] THEN
									IF Mach_Control.WJ_b.SinStepMode THEN//尾卷单步模式
										TailCurlSinStep:=TRUE;
									ELSE
										TailCurlSinStep:=FALSE;
									END_IF	
									TailCurlStep3:=140;
								END_IF
						END_IF
				140://左、右压刀开合轴至张开位
						IF NOT TailCurlSinStep THEN					
								IF 	arrAxisCtrl[AxiseNo.AxisName.LeftYDLine].Status.Homed AND arrAxisCtrl[AxiseNo.AxisName.LeftYDLine].Status.NoMoving THEN
									IF arrAxisCtrl[AxiseNo.AxisName.LeftYDLine].Cmd.arrbRealPoint[2] THEN
										arrAxisCtrl[AxiseNo.AxisName.LeftYDLine].Cmd.iGoSetPos:=0;
									ELSE
										arrAxisCtrl[AxiseNo.AxisName.LeftYDLine].Cmd.iGoSetPos:=2;//左压刀开合至张开位
									END_IF
								END_IF					
								IF 	arrAxisCtrl[AxiseNo.AxisName.RightYDLine].Status.Homed AND arrAxisCtrl[AxiseNo.AxisName.RightYDLine].Status.NoMoving THEN
									IF arrAxisCtrl[AxiseNo.AxisName.RightYDLine].Cmd.arrbRealPoint[3] THEN
										arrAxisCtrl[AxiseNo.AxisName.RightYDLine].Cmd.iGoSetPos:=0;
									ELSE
										arrAxisCtrl[AxiseNo.AxisName.RightYDLine].Cmd.iGoSetPos:=3;//右压刀开合至张开位
									END_IF
								END_IF				
								IF arrAxisCtrl[AxiseNo.AxisName.LeftYDLine].Cmd.arrbRealPoint[2] AND arrAxisCtrl[AxiseNo.AxisName.RightYDLine].Cmd.arrbRealPoint[3] THEN
									IF Mach_Control.WJ_b.SinStepMode THEN//尾卷单步模式
										TailCurlSinStep:=TRUE;
									ELSE
										TailCurlSinStep:=FALSE;
									END_IF										
									TailCurlStep3:=145;
								END_IF	
						END_IF
						
				145:
						IF NOT TailCurlSinStep THEN		
								IF 	arrAxisCtrl[AxiseNo.AxisName.RightYDUpDown].Status.Homed AND arrAxisCtrl[AxiseNo.AxisName.RightYDUpDown].Status.NoMoving THEN
									IF arrAxisCtrl[AxiseNo.AxisName.RightYDUpDown].Cmd.arrbRealPoint[5] THEN
										arrAxisCtrl[AxiseNo.AxisName.RightYDUpDown].Cmd.iGoSetPos:=0;
									ELSE
										arrAxisCtrl[AxiseNo.AxisName.RightYDUpDown].Cmd.iGoSetPos:=5;//右压好升降上升至下料张开位
									END_IF
								END_IF				
								IF  arrAxisCtrl[AxiseNo.AxisName.RightYDUpDown].Cmd.arrbRealPoint[5] THEN
									IF Mach_Control.WJ_b.SinStepMode THEN//尾卷单步模式
										TailCurlSinStep:=TRUE;
									ELSE
										TailCurlSinStep:=FALSE;
									END_IF	
									TailCurlStep3:=150;
								END_IF

						END_IF
		
						
				146:
				
					(*IF NOT TailCurlSinStep THEN	
								arrCyCtrl[arrCyNo.CylinderName.PreDiaph].Cmd.bON:=TRUE;//叠台压隔膜气缸
								IF arrCyCtrl[arrCyNo.CylinderName.PreDiaph].Io.DIOnSwitch THEN
											IF Mach_Control.WJ_b.SinStepMode THEN//尾卷单步模式
												TailCurlSinStep:=TRUE;
											ELSE
												TailCurlSinStep:=FALSE;
											END_IF							
											TailCurlStep3:=150;	
								END_IF	
					END_IF*)	
						
						
				150://尾卷夹电芯平移至拉膜位、尾卷夹电芯伸缩至初始位、
						IF NOT TailCurlSinStep THEN	
							tailCult_GearInMultiMaster.Enable:=TRUE;//启动尾卷拉膜凸轮耦合
							fbGearInGMvirbEnable:=TRUE;//尾卷拉膜纠偏
							//Par.stDT_date.iTargetTorqueBLXS:=6;
							IF  tailCult_GearInMultiMaster.InGear THEN
								
										IF arrAxisCtrl[AxiseNo.AxisName.TailCurlLine].Status.fActPos<LREAL_TO_REAL(arrAxispar[AxiseNo.AxisName.TailCurlLine].arrTargetPoint[3]+100) THEN
											arrAxisCtrl[AxiseNo.AxisName.TailCurlLine].Cmd.fOverride:=60;
										END_IF
										IF 	arrAxisCtrl[AxiseNo.AxisName.TailCurlRetracting].Status.Homed AND arrAxisCtrl[AxiseNo.AxisName.TailCurlRetracting].Status.NoMoving AND
                                                arrAxisCtrl[AxiseNo.AxisName.LCurlingneedleLine].Cmd.arrbRealPoint[1]  AND arrAxisCtrl[AxiseNo.AxisName.SCurlingneedleLine].Cmd.arrbRealPoint[1]  THEN
										
